% RSLogix 500 project VENTURA PACIFIC 3D_BAK170.RSS, saved by version 11.00.00.00 %
PROJECT "UNTITLED"    % processor: MicroLogix 1400 %

PROGRAM FILES
  LAD 2   213 rungs

DATA FILES
  O0 OUTPUT  7 elements
  I1 INPUT  26 elements
  S2 STATUS  66 elements
  B3 BINARY  10 elements
  T4 TIMER  35 elements  % Moves timing value into Time delay for bin eject %
  C5 COUNTER  9 elements
  R6 CONTROL  1 elements
  N7 INTEGER  33 elements
  F8 FLOAT  3 elements

LADDER 2
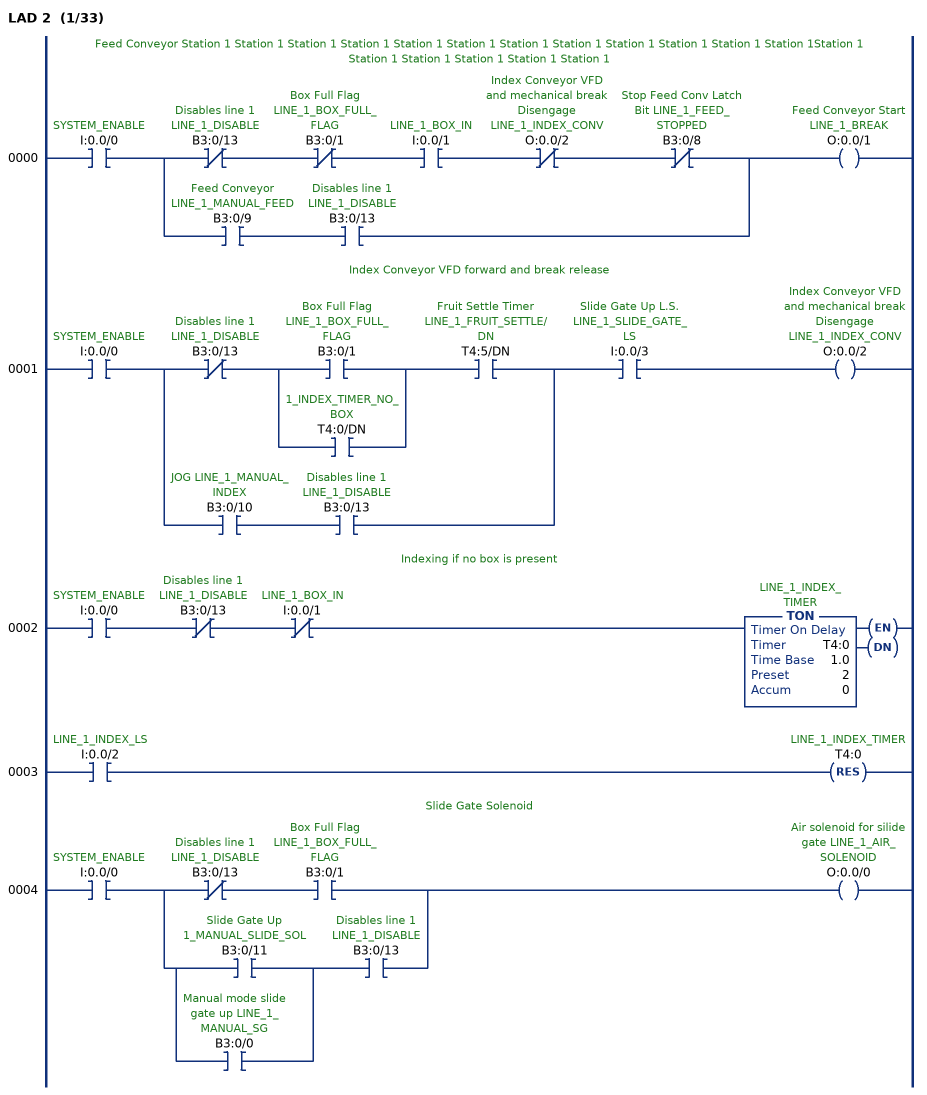
% Rung: 0 %
% Feed Conveyor Station 1 Station 1 Station 1 Station 1 Station 1 Station 1 Station 1 Station 1 Station 1 Station 1 Station 1 Station 1Station 1 Station 1 Station 1 Station 1 Station 1 Station 1 %
SOR XIC I:0.0/0 BST XIO B3:0/13 XIO B3:0/1 XIC I:0.0/1 XIO O:0.0/2 XIO B3:0/8 NXB XIC B3:0/9 XIC B3:0/13 BND OTE O:0.0/1 EOR
%   I:0.0/0  SYSTEM_ENABLE %
%   B3:0/13  LINE_1_DISABLE  "Disables line 1" %
%   B3:0/1  LINE_1_BOX_FULL_FLAG  "Box Full Flag" %
%   I:0.0/1  LINE_1_BOX_IN %
%   O:0.0/2  LINE_1_INDEX_CONV  "Index Conveyor VFD and mechanical break Disengage" %
%   B3:0/8  LINE_1_FEED_STOPPED  "Stop Feed Conv Latch Bit" %
%   B3:0/9  LINE_1_MANUAL_FEED  "Feed Conveyor" %
%   O:0.0/1  LINE_1_BREAK  "Feed Conveyor Start" %
% Rung: 1 %
% Index Conveyor VFD forward and break release %
SOR XIC I:0.0/0 BST XIO B3:0/13 BST XIC B3:0/1 NXB XIC T4:0/DN BND XIC T4:5/DN NXB XIC B3:0/10 XIC B3:0/13 BND XIC I:0.0/3 OTE O:0.0/2 EOR
%   I:0.0/0  SYSTEM_ENABLE %
%   B3:0/13  LINE_1_DISABLE  "Disables line 1" %
%   B3:0/1  LINE_1_BOX_FULL_FLAG  "Box Full Flag" %
%   T4:0/DN  1_INDEX_TIMER_NO_BOX %
%   T4:5  LINE_1_FRUIT_SETTLE  "Fruit Settle Timer" %
%   B3:0/10  LINE_1_MANUAL_INDEX  "JOG" %
%   I:0.0/3  LINE_1_SLIDE_GATE_LS  "Slide Gate Up L.S." %
%   O:0.0/2  LINE_1_INDEX_CONV  "Index Conveyor VFD and mechanical break Disengage" %
% Rung: 2 %
% Indexing if no box is present %
SOR XIC I:0.0/0 XIO B3:0/13 XIO I:0.0/1 TON T4:0 1.0 2 0 EOR
%   I:0.0/0  SYSTEM_ENABLE %
%   B3:0/13  LINE_1_DISABLE  "Disables line 1" %
%   I:0.0/1  LINE_1_BOX_IN %
%   T4:0  LINE_1_INDEX_TIMER %
% Rung: 3 %
SOR XIC I:0.0/2 RES T4:0 EOR
%   I:0.0/2  LINE_1_INDEX_LS %
%   T4:0  LINE_1_INDEX_TIMER %
% Rung: 4 %
% Slide Gate Solenoid %
SOR XIC I:0.0/0 BST XIO B3:0/13 XIC B3:0/1 NXB BST XIC B3:0/11 NXB XIC B3:0/0 BND XIC B3:0/13 BND OTE O:0.0/0 EOR
%   I:0.0/0  SYSTEM_ENABLE %
%   B3:0/13  LINE_1_DISABLE  "Disables line 1" %
%   B3:0/1  LINE_1_BOX_FULL_FLAG  "Box Full Flag" %
%   B3:0/11  1_MANUAL_SLIDE_SOL  "Slide Gate Up" %
%   B3:0/0  LINE_1_MANUAL_SG  "Manual mode slide gate up" %
%   O:0.0/0  LINE_1_AIR_SOLENOID  "Air solenoid for silide gate" %

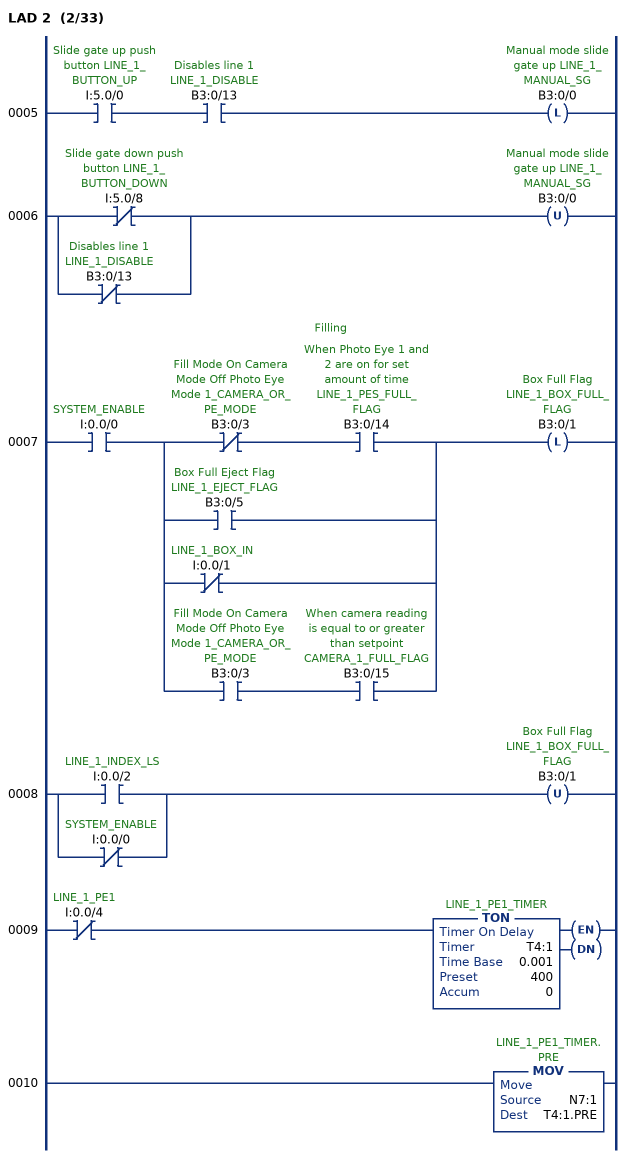
% Rung: 5 %
SOR XIC I:5.0/0 XIC B3:0/13 OTL B3:0/0 EOR
%   I:5.0/0  LINE_1_BUTTON_UP  "Slide gate up push button" %
%   B3:0/13  LINE_1_DISABLE  "Disables line 1" %
%   B3:0/0  LINE_1_MANUAL_SG  "Manual mode slide gate up" %
% Rung: 6 %
SOR BST XIO I:5.0/8 NXB XIO B3:0/13 BND OTU B3:0/0 EOR
%   I:5.0/8  LINE_1_BUTTON_DOWN  "Slide gate down push button" %
%   B3:0/13  LINE_1_DISABLE  "Disables line 1" %
%   B3:0/0  LINE_1_MANUAL_SG  "Manual mode slide gate up" %
% Rung: 7 %
% Filling %
SOR XIC I:0.0/0 BST XIO B3:0/3 XIC B3:0/14 NXB BST XIC B3:0/5 NXB BST XIO I:0.0/1 NXB XIC B3:0/3 XIC B3:0/15 BND BND BND OTL B3:0/1 EOR
%   I:0.0/0  SYSTEM_ENABLE %
%   B3:0/3  1_CAMERA_OR_PE_MODE  "Fill Mode On Camera Mode Off Photo Eye Mode" %
%   B3:0/14  LINE_1_PES_FULL_FLAG  "When Photo Eye 1 and 2 are on for set amount of time" %
%   B3:0/5  LINE_1_EJECT_FLAG  "Box Full Eject Flag" %
%   I:0.0/1  LINE_1_BOX_IN %
%   B3:0/15  CAMERA_1_FULL_FLAG  "When camera reading is equal to or greater than setpoint" %
%   B3:0/1  LINE_1_BOX_FULL_FLAG  "Box Full Flag" %
% Rung: 8 %
SOR BST XIC I:0.0/2 NXB XIO I:0.0/0 BND OTU B3:0/1 EOR
%   I:0.0/2  LINE_1_INDEX_LS %
%   I:0.0/0  SYSTEM_ENABLE %
%   B3:0/1  LINE_1_BOX_FULL_FLAG  "Box Full Flag" %
% Rung: 9 %
SOR XIO I:0.0/4 TON T4:1 0.001 400 0 EOR
%   I:0.0/4  LINE_1_PE1 %
%   T4:1  LINE_1_PE1_TIMER %
% Rung: 10 %
SOR MOV N7:1 T4:1.PRE EOR
%   N7:1  LINE_1_PE1_TIME_MOV %
%   T4:1  LINE_1_PE1_TIMER %

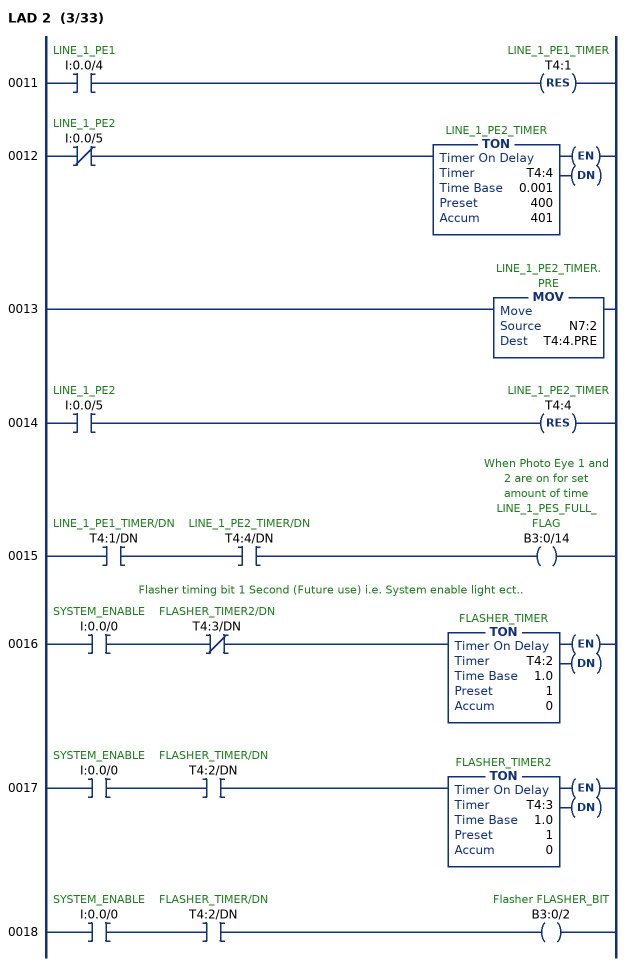
% Rung: 11 %
SOR XIC I:0.0/4 RES T4:1 EOR
%   I:0.0/4  LINE_1_PE1 %
%   T4:1  LINE_1_PE1_TIMER %
% Rung: 12 %
SOR XIO I:0.0/5 TON T4:4 0.001 400 401 EOR
%   I:0.0/5  LINE_1_PE2 %
%   T4:4  LINE_1_PE2_TIMER %
% Rung: 13 %
SOR MOV N7:2 T4:4.PRE EOR
%   N7:2  LINE_1_PE2_TIME_MOV %
%   T4:4  LINE_1_PE2_TIMER %
% Rung: 14 %
SOR XIC I:0.0/5 RES T4:4 EOR
%   I:0.0/5  LINE_1_PE2 %
%   T4:4  LINE_1_PE2_TIMER %
% Rung: 15 %
SOR XIC T4:1/DN XIC T4:4/DN OTE B3:0/14 EOR
%   T4:1  LINE_1_PE1_TIMER %
%   T4:4  LINE_1_PE2_TIMER %
%   B3:0/14  LINE_1_PES_FULL_FLAG  "When Photo Eye 1 and 2 are on for set amount of time" %
% Rung: 16 %
% Flasher timing bit 1 Second (Future use) i.e. System enable light ect.. %
SOR XIC I:0.0/0 XIO T4:3/DN TON T4:2 1.0 1 0 EOR
%   I:0.0/0  SYSTEM_ENABLE %
%   T4:3  FLASHER_TIMER2 %
%   T4:2  FLASHER_TIMER %
% Rung: 17 %
SOR XIC I:0.0/0 XIC T4:2/DN TON T4:3 1.0 1 0 EOR
%   I:0.0/0  SYSTEM_ENABLE %
%   T4:2  FLASHER_TIMER %
%   T4:3  FLASHER_TIMER2 %
% Rung: 18 %
SOR XIC I:0.0/0 XIC T4:2/DN OTE B3:0/2 EOR
%   I:0.0/0  SYSTEM_ENABLE %
%   T4:2  FLASHER_TIMER %
%   B3:0/2  FLASHER_BIT  "Flasher" %

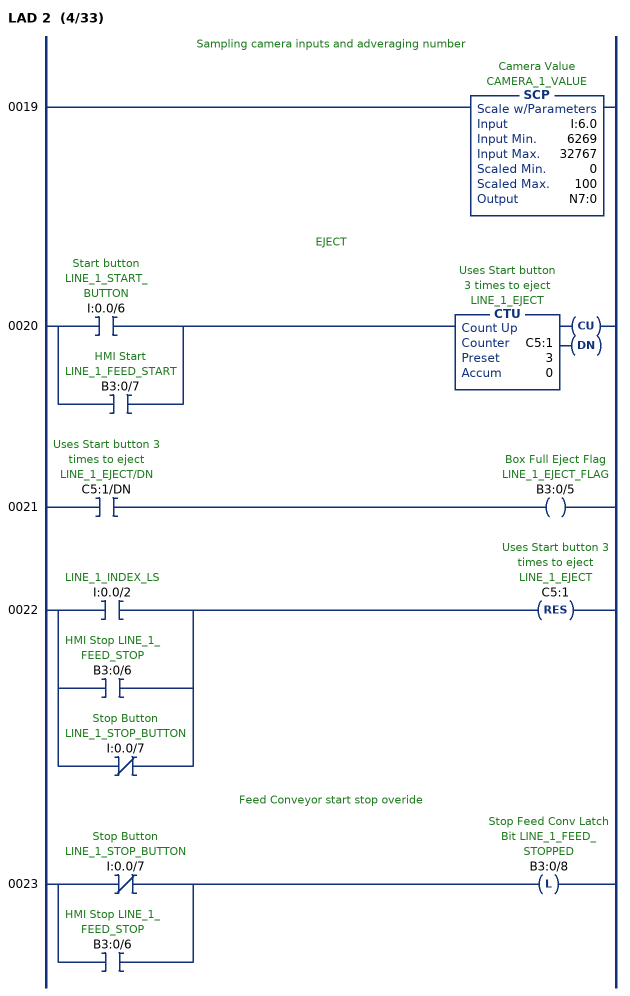
% Rung: 19 %
% Sampling camera inputs and adveraging number %
SOR SCP I:6.0 6269 32767 0 100 N7:0 EOR
%   N7:0  CAMERA_1_VALUE  "Camera Value" %
% Rung: 20 %
% EJECT %
SOR BST XIC I:0.0/6 NXB XIC B3:0/7 BND CTU C5:1 3 0 EOR
%   I:0.0/6  LINE_1_START_BUTTON  "Start button" %
%   B3:0/7  LINE_1_FEED_START  "HMI Start" %
%   C5:1  LINE_1_EJECT  "Uses Start button 3 times to eject" %
% Rung: 21 %
SOR XIC C5:1/DN OTE B3:0/5 EOR
%   C5:1  LINE_1_EJECT  "Uses Start button 3 times to eject" %
%   B3:0/5  LINE_1_EJECT_FLAG  "Box Full Eject Flag" %
% Rung: 22 %
SOR BST XIC I:0.0/2 NXB BST XIC B3:0/6 NXB XIO I:0.0/7 BND BND RES C5:1 EOR
%   I:0.0/2  LINE_1_INDEX_LS %
%   B3:0/6  LINE_1_FEED_STOP  "HMI Stop" %
%   I:0.0/7  LINE_1_STOP_BUTTON  "Stop Button" %
%   C5:1  LINE_1_EJECT  "Uses Start button 3 times to eject" %
% Rung: 23 %
% Feed Conveyor start stop overide %
SOR BST XIO I:0.0/7 NXB XIC B3:0/6 BND OTL B3:0/8 EOR
%   I:0.0/7  LINE_1_STOP_BUTTON  "Stop Button" %
%   B3:0/6  LINE_1_FEED_STOP  "HMI Stop" %
%   B3:0/8  LINE_1_FEED_STOPPED  "Stop Feed Conv Latch Bit" %

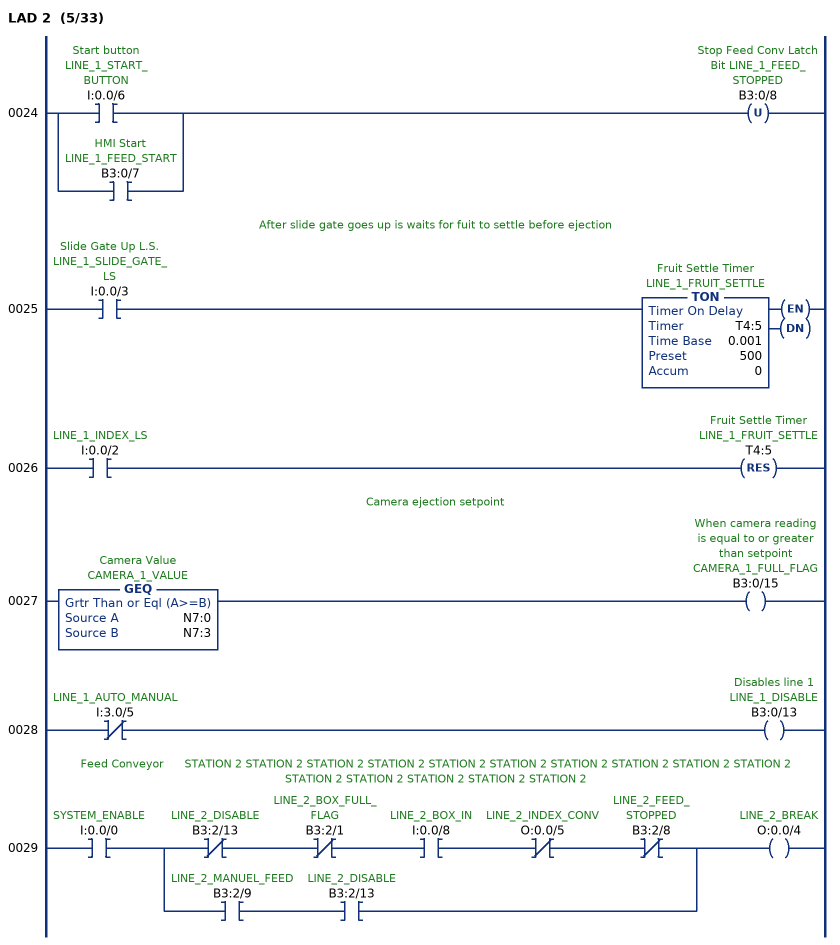
% Rung: 24 %
SOR BST XIC I:0.0/6 NXB XIC B3:0/7 BND OTU B3:0/8 EOR
%   I:0.0/6  LINE_1_START_BUTTON  "Start button" %
%   B3:0/7  LINE_1_FEED_START  "HMI Start" %
%   B3:0/8  LINE_1_FEED_STOPPED  "Stop Feed Conv Latch Bit" %
% Rung: 25 %
% After slide gate goes up is waits for fuit to settle before ejection %
SOR XIC I:0.0/3 TON T4:5 0.001 500 0 EOR
%   I:0.0/3  LINE_1_SLIDE_GATE_LS  "Slide Gate Up L.S." %
%   T4:5  LINE_1_FRUIT_SETTLE  "Fruit Settle Timer" %
% Rung: 26 %
SOR XIC I:0.0/2 RES T4:5 EOR
%   I:0.0/2  LINE_1_INDEX_LS %
%   T4:5  LINE_1_FRUIT_SETTLE  "Fruit Settle Timer" %
% Rung: 27 %
% Camera ejection setpoint %
SOR GEQ N7:0 N7:3 OTE B3:0/15 EOR
%   N7:0  CAMERA_1_VALUE  "Camera Value" %
%   N7:3  LINE_1_CAMERA_EJECT %
%   B3:0/15  CAMERA_1_FULL_FLAG  "When camera reading is equal to or greater than setpoint" %
% Rung: 28 %
SOR XIO I:3.0/5 OTE B3:0/13 EOR
%   I:3.0/5  LINE_1_AUTO_MANUAL %
%   B3:0/13  LINE_1_DISABLE  "Disables line 1" %
% Rung: 29 %
% Feed Conveyor      STATION 2 STATION 2 STATION 2 STATION 2 STATION 2 STATION 2 STATION 2 STATION 2 STATION 2 STATION 2 STATION 2 STATION 2 STATION 2 STATION 2 STATION 2 %
SOR XIC I:0.0/0 BST XIO B3:2/13 XIO B3:2/1 XIC I:0.0/8 XIO O:0.0/5 XIO B3:2/8 NXB XIC B3:2/9 XIC B3:2/13 BND OTE O:0.0/4 EOR
%   I:0.0/0  SYSTEM_ENABLE %
%   B3:2/13  LINE_2_DISABLE %
%   B3:2/1  LINE_2_BOX_FULL_FLAG %
%   I:0.0/8  LINE_2_BOX_IN %
%   O:0.0/5  LINE_2_INDEX_CONV %
%   B3:2/8  LINE_2_FEED_STOPPED %
%   B3:2/9  LINE_2_MANUEL_FEED %
%   O:0.0/4  LINE_2_BREAK %

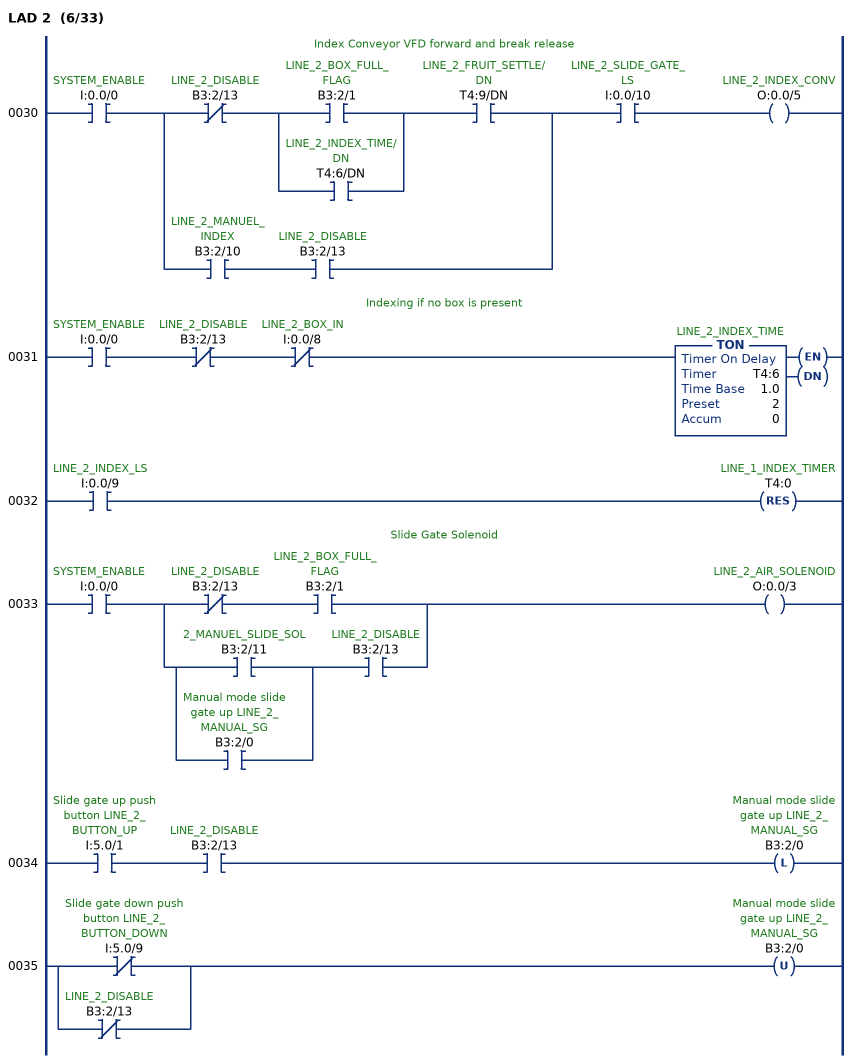
% Rung: 30 %
% Index Conveyor VFD forward and break release %
SOR XIC I:0.0/0 BST XIO B3:2/13 BST XIC B3:2/1 NXB XIC T4:6/DN BND XIC T4:9/DN NXB XIC B3:2/10 XIC B3:2/13 BND XIC I:0.0/10 OTE O:0.0/5 EOR
%   I:0.0/0  SYSTEM_ENABLE %
%   B3:2/13  LINE_2_DISABLE %
%   B3:2/1  LINE_2_BOX_FULL_FLAG %
%   T4:6  LINE_2_INDEX_TIME %
%   T4:9  LINE_2_FRUIT_SETTLE %
%   B3:2/10  LINE_2_MANUEL_INDEX %
%   I:0.0/10  LINE_2_SLIDE_GATE_LS %
%   O:0.0/5  LINE_2_INDEX_CONV %
% Rung: 31 %
% Indexing if no box is present %
SOR XIC I:0.0/0 XIO B3:2/13 XIO I:0.0/8 TON T4:6 1.0 2 0 EOR
%   I:0.0/0  SYSTEM_ENABLE %
%   B3:2/13  LINE_2_DISABLE %
%   I:0.0/8  LINE_2_BOX_IN %
%   T4:6  LINE_2_INDEX_TIME %
% Rung: 32 %
SOR XIC I:0.0/9 RES T4:0 EOR
%   I:0.0/9  LINE_2_INDEX_LS %
%   T4:0  LINE_1_INDEX_TIMER %
% Rung: 33 %
% Slide Gate Solenoid %
SOR XIC I:0.0/0 BST XIO B3:2/13 XIC B3:2/1 NXB BST XIC B3:2/11 NXB XIC B3:2/0 BND XIC B3:2/13 BND OTE O:0.0/3 EOR
%   I:0.0/0  SYSTEM_ENABLE %
%   B3:2/13  LINE_2_DISABLE %
%   B3:2/1  LINE_2_BOX_FULL_FLAG %
%   B3:2/11  2_MANUEL_SLIDE_SOL %
%   B3:2/0  LINE_2_MANUAL_SG  "Manual mode slide gate up" %
%   O:0.0/3  LINE_2_AIR_SOLENOID %
% Rung: 34 %
SOR XIC I:5.0/1 XIC B3:2/13 OTL B3:2/0 EOR
%   I:5.0/1  LINE_2_BUTTON_UP  "Slide gate up push button" %
%   B3:2/13  LINE_2_DISABLE %
%   B3:2/0  LINE_2_MANUAL_SG  "Manual mode slide gate up" %
% Rung: 35 %
SOR BST XIO I:5.0/9 NXB XIO B3:2/13 BND OTU B3:2/0 EOR
%   I:5.0/9  LINE_2_BUTTON_DOWN  "Slide gate down push button" %
%   B3:2/13  LINE_2_DISABLE %
%   B3:2/0  LINE_2_MANUAL_SG  "Manual mode slide gate up" %

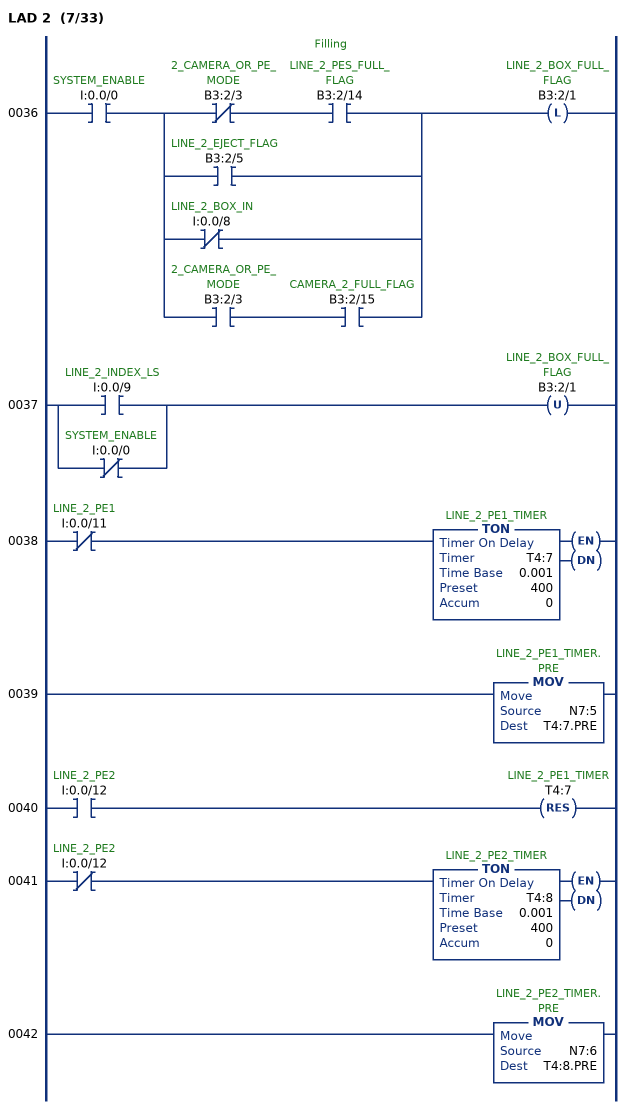
% Rung: 36 %
% Filling %
SOR XIC I:0.0/0 BST XIO B3:2/3 XIC B3:2/14 NXB BST XIC B3:2/5 NXB BST XIO I:0.0/8 NXB XIC B3:2/3 XIC B3:2/15 BND BND BND OTL B3:2/1 EOR
%   I:0.0/0  SYSTEM_ENABLE %
%   B3:2/3  2_CAMERA_OR_PE_MODE %
%   B3:2/14  LINE_2_PES_FULL_FLAG %
%   B3:2/5  LINE_2_EJECT_FLAG %
%   I:0.0/8  LINE_2_BOX_IN %
%   B3:2/15  CAMERA_2_FULL_FLAG %
%   B3:2/1  LINE_2_BOX_FULL_FLAG %
% Rung: 37 %
SOR BST XIC I:0.0/9 NXB XIO I:0.0/0 BND OTU B3:2/1 EOR
%   I:0.0/9  LINE_2_INDEX_LS %
%   I:0.0/0  SYSTEM_ENABLE %
%   B3:2/1  LINE_2_BOX_FULL_FLAG %
% Rung: 38 %
SOR XIO I:0.0/11 TON T4:7 0.001 400 0 EOR
%   I:0.0/11  LINE_2_PE1 %
%   T4:7  LINE_2_PE1_TIMER %
% Rung: 39 %
SOR MOV N7:5 T4:7.PRE EOR
%   N7:5  LINE_2_PE1_TIME_MOV %
%   T4:7  LINE_2_PE1_TIMER %
% Rung: 40 %
SOR XIC I:0.0/12 RES T4:7 EOR
%   I:0.0/12  LINE_2_PE2 %
%   T4:7  LINE_2_PE1_TIMER %
% Rung: 41 %
SOR XIO I:0.0/12 TON T4:8 0.001 400 0 EOR
%   I:0.0/12  LINE_2_PE2 %
%   T4:8  LINE_2_PE2_TIMER %
% Rung: 42 %
SOR MOV N7:6 T4:8.PRE EOR
%   N7:6  LINE_2_PE2_TIME_MOV %
%   T4:8  LINE_2_PE2_TIMER %

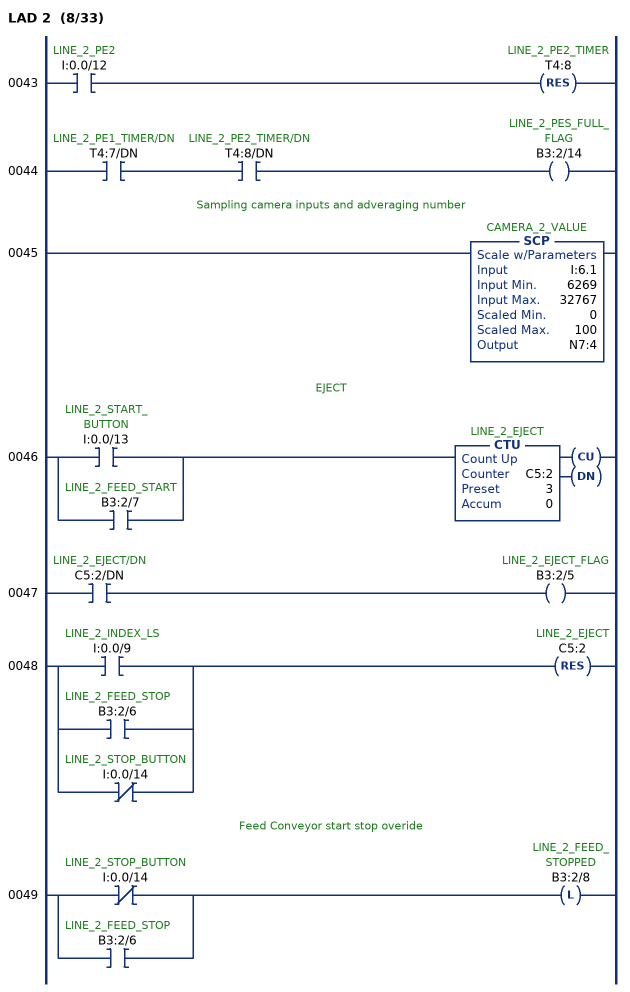
% Rung: 43 %
SOR XIC I:0.0/12 RES T4:8 EOR
%   I:0.0/12  LINE_2_PE2 %
%   T4:8  LINE_2_PE2_TIMER %
% Rung: 44 %
SOR XIC T4:7/DN XIC T4:8/DN OTE B3:2/14 EOR
%   T4:7  LINE_2_PE1_TIMER %
%   T4:8  LINE_2_PE2_TIMER %
%   B3:2/14  LINE_2_PES_FULL_FLAG %
% Rung: 45 %
% Sampling camera inputs and adveraging number %
SOR SCP I:6.1 6269 32767 0 100 N7:4 EOR
%   N7:4  CAMERA_2_VALUE %
% Rung: 46 %
% EJECT %
SOR BST XIC I:0.0/13 NXB XIC B3:2/7 BND CTU C5:2 3 0 EOR
%   I:0.0/13  LINE_2_START_BUTTON %
%   B3:2/7  LINE_2_FEED_START %
%   C5:2  LINE_2_EJECT %
% Rung: 47 %
SOR XIC C5:2/DN OTE B3:2/5 EOR
%   C5:2  LINE_2_EJECT %
%   B3:2/5  LINE_2_EJECT_FLAG %
% Rung: 48 %
SOR BST XIC I:0.0/9 NXB BST XIC B3:2/6 NXB XIO I:0.0/14 BND BND RES C5:2 EOR
%   I:0.0/9  LINE_2_INDEX_LS %
%   B3:2/6  LINE_2_FEED_STOP %
%   I:0.0/14  LINE_2_STOP_BUTTON %
%   C5:2  LINE_2_EJECT %
% Rung: 49 %
% Feed Conveyor start stop overide %
SOR BST XIO I:0.0/14 NXB XIC B3:2/6 BND OTL B3:2/8 EOR
%   I:0.0/14  LINE_2_STOP_BUTTON %
%   B3:2/6  LINE_2_FEED_STOP %
%   B3:2/8  LINE_2_FEED_STOPPED %

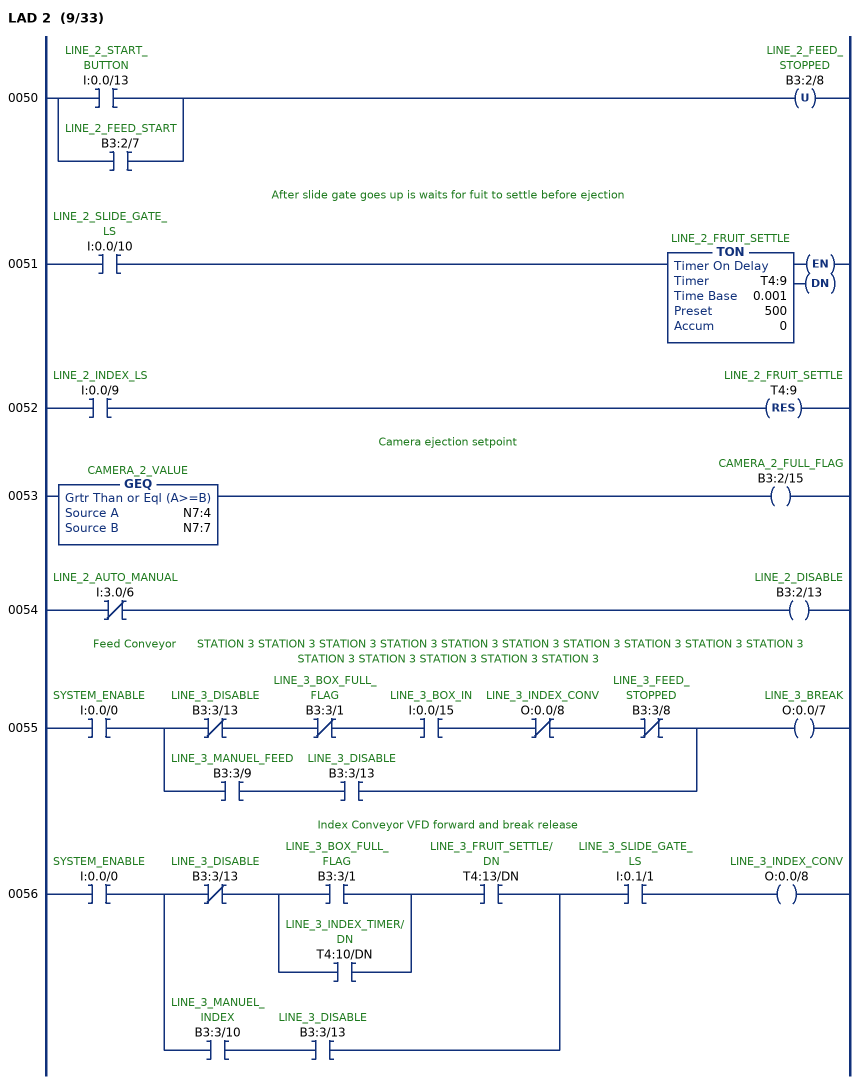
% Rung: 50 %
SOR BST XIC I:0.0/13 NXB XIC B3:2/7 BND OTU B3:2/8 EOR
%   I:0.0/13  LINE_2_START_BUTTON %
%   B3:2/7  LINE_2_FEED_START %
%   B3:2/8  LINE_2_FEED_STOPPED %
% Rung: 51 %
% After slide gate goes up is waits for fuit to settle before ejection %
SOR XIC I:0.0/10 TON T4:9 0.001 500 0 EOR
%   I:0.0/10  LINE_2_SLIDE_GATE_LS %
%   T4:9  LINE_2_FRUIT_SETTLE %
% Rung: 52 %
SOR XIC I:0.0/9 RES T4:9 EOR
%   I:0.0/9  LINE_2_INDEX_LS %
%   T4:9  LINE_2_FRUIT_SETTLE %
% Rung: 53 %
% Camera ejection setpoint %
SOR GEQ N7:4 N7:7 OTE B3:2/15 EOR
%   N7:4  CAMERA_2_VALUE %
%   N7:7  LINE_2_CAMERA_EJECT %
%   B3:2/15  CAMERA_2_FULL_FLAG %
% Rung: 54 %
SOR XIO I:3.0/6 OTE B3:2/13 EOR
%   I:3.0/6  LINE_2_AUTO_MANUAL %
%   B3:2/13  LINE_2_DISABLE %
% Rung: 55 %
% Feed Conveyor      STATION 3 STATION 3 STATION 3 STATION 3 STATION 3 STATION 3 STATION 3 STATION 3 STATION 3 STATION 3 STATION 3 STATION 3 STATION 3 STATION 3 STATION 3 %
SOR XIC I:0.0/0 BST XIO B3:3/13 XIO B3:3/1 XIC I:0.0/15 XIO O:0.0/8 XIO B3:3/8 NXB XIC B3:3/9 XIC B3:3/13 BND OTE O:0.0/7 EOR
%   I:0.0/0  SYSTEM_ENABLE %
%   B3:3/13  LINE_3_DISABLE %
%   B3:3/1  LINE_3_BOX_FULL_FLAG %
%   I:0.0/15  LINE_3_BOX_IN %
%   O:0.0/8  LINE_3_INDEX_CONV %
%   B3:3/8  LINE_3_FEED_STOPPED %
%   B3:3/9  LINE_3_MANUEL_FEED %
%   O:0.0/7  LINE_3_BREAK %
% Rung: 56 %
% Index Conveyor VFD forward and break release %
SOR XIC I:0.0/0 BST XIO B3:3/13 BST XIC B3:3/1 NXB XIC T4:10/DN BND XIC T4:13/DN NXB XIC B3:3/10 XIC B3:3/13 BND XIC I:0.1/1 OTE O:0.0/8 EOR
%   I:0.0/0  SYSTEM_ENABLE %
%   B3:3/13  LINE_3_DISABLE %
%   B3:3/1  LINE_3_BOX_FULL_FLAG %
%   T4:10  LINE_3_INDEX_TIMER %
%   T4:13  LINE_3_FRUIT_SETTLE %
%   B3:3/10  LINE_3_MANUEL_INDEX %
%   I:0.1/1  LINE_3_SLIDE_GATE_LS %
%   O:0.0/8  LINE_3_INDEX_CONV %

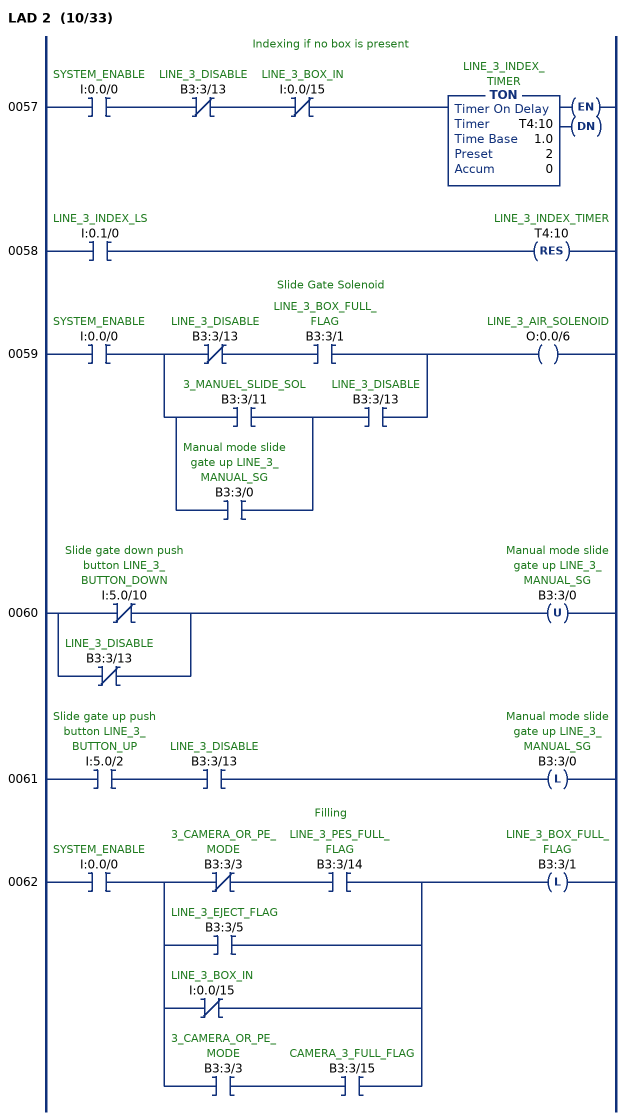
% Rung: 57 %
% Indexing if no box is present %
SOR XIC I:0.0/0 XIO B3:3/13 XIO I:0.0/15 TON T4:10 1.0 2 0 EOR
%   I:0.0/0  SYSTEM_ENABLE %
%   B3:3/13  LINE_3_DISABLE %
%   I:0.0/15  LINE_3_BOX_IN %
%   T4:10  LINE_3_INDEX_TIMER %
% Rung: 58 %
SOR XIC I:0.1/0 RES T4:10 EOR
%   I:0.1/0  LINE_3_INDEX_LS %
%   T4:10  LINE_3_INDEX_TIMER %
% Rung: 59 %
% Slide Gate Solenoid %
SOR XIC I:0.0/0 BST XIO B3:3/13 XIC B3:3/1 NXB BST XIC B3:3/11 NXB XIC B3:3/0 BND XIC B3:3/13 BND OTE O:0.0/6 EOR
%   I:0.0/0  SYSTEM_ENABLE %
%   B3:3/13  LINE_3_DISABLE %
%   B3:3/1  LINE_3_BOX_FULL_FLAG %
%   B3:3/11  3_MANUEL_SLIDE_SOL %
%   B3:3/0  LINE_3_MANUAL_SG  "Manual mode slide gate up" %
%   O:0.0/6  LINE_3_AIR_SOLENOID %
% Rung: 60 %
SOR BST XIO I:5.0/10 NXB XIO B3:3/13 BND OTU B3:3/0 EOR
%   I:5.0/10  LINE_3_BUTTON_DOWN  "Slide gate down push button" %
%   B3:3/13  LINE_3_DISABLE %
%   B3:3/0  LINE_3_MANUAL_SG  "Manual mode slide gate up" %
% Rung: 61 %
SOR XIC I:5.0/2 XIC B3:3/13 OTL B3:3/0 EOR
%   I:5.0/2  LINE_3_BUTTON_UP  "Slide gate up push button" %
%   B3:3/13  LINE_3_DISABLE %
%   B3:3/0  LINE_3_MANUAL_SG  "Manual mode slide gate up" %
% Rung: 62 %
% Filling %
SOR XIC I:0.0/0 BST XIO B3:3/3 XIC B3:3/14 NXB BST XIC B3:3/5 NXB BST XIO I:0.0/15 NXB XIC B3:3/3 XIC B3:3/15 BND BND BND OTL B3:3/1 EOR
%   I:0.0/0  SYSTEM_ENABLE %
%   B3:3/3  3_CAMERA_OR_PE_MODE %
%   B3:3/14  LINE_3_PES_FULL_FLAG %
%   B3:3/5  LINE_3_EJECT_FLAG %
%   I:0.0/15  LINE_3_BOX_IN %
%   B3:3/15  CAMERA_3_FULL_FLAG %
%   B3:3/1  LINE_3_BOX_FULL_FLAG %

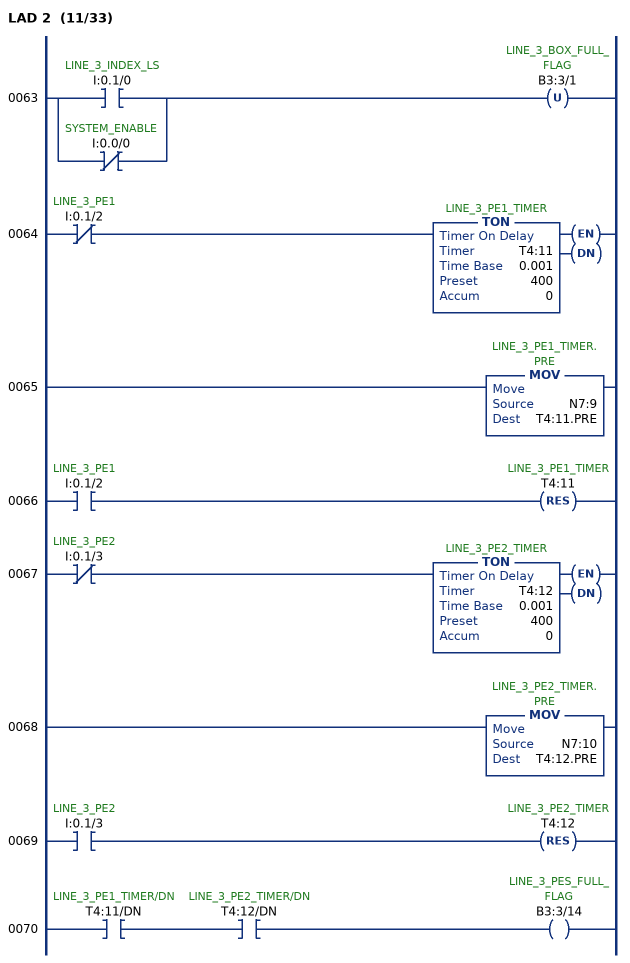
% Rung: 63 %
SOR BST XIC I:0.1/0 NXB XIO I:0.0/0 BND OTU B3:3/1 EOR
%   I:0.1/0  LINE_3_INDEX_LS %
%   I:0.0/0  SYSTEM_ENABLE %
%   B3:3/1  LINE_3_BOX_FULL_FLAG %
% Rung: 64 %
SOR XIO I:0.1/2 TON T4:11 0.001 400 0 EOR
%   I:0.1/2  LINE_3_PE1 %
%   T4:11  LINE_3_PE1_TIMER %
% Rung: 65 %
SOR MOV N7:9 T4:11.PRE EOR
%   N7:9  LINE_3_PE1_TIME_MOV %
%   T4:11  LINE_3_PE1_TIMER %
% Rung: 66 %
SOR XIC I:0.1/2 RES T4:11 EOR
%   I:0.1/2  LINE_3_PE1 %
%   T4:11  LINE_3_PE1_TIMER %
% Rung: 67 %
SOR XIO I:0.1/3 TON T4:12 0.001 400 0 EOR
%   I:0.1/3  LINE_3_PE2 %
%   T4:12  LINE_3_PE2_TIMER %
% Rung: 68 %
SOR MOV N7:10 T4:12.PRE EOR
%   N7:10  LINE_3_PE2_TIME_MOV %
%   T4:12  LINE_3_PE2_TIMER %
% Rung: 69 %
SOR XIC I:0.1/3 RES T4:12 EOR
%   I:0.1/3  LINE_3_PE2 %
%   T4:12  LINE_3_PE2_TIMER %
% Rung: 70 %
SOR XIC T4:11/DN XIC T4:12/DN OTE B3:3/14 EOR
%   T4:11  LINE_3_PE1_TIMER %
%   T4:12  LINE_3_PE2_TIMER %
%   B3:3/14  LINE_3_PES_FULL_FLAG %

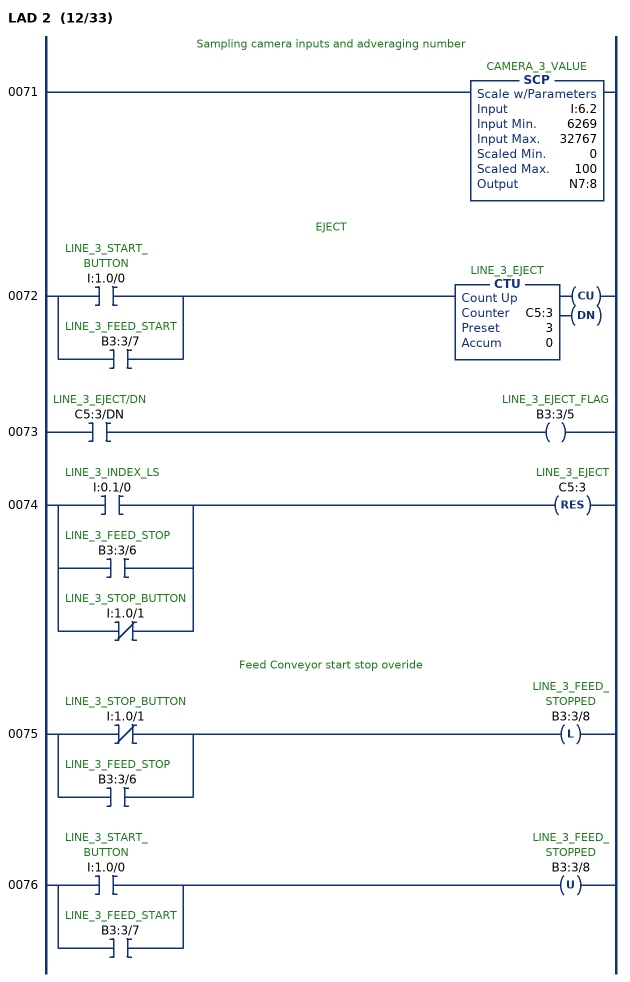
% Rung: 71 %
% Sampling camera inputs and adveraging number %
SOR SCP I:6.2 6269 32767 0 100 N7:8 EOR
%   N7:8  CAMERA_3_VALUE %
% Rung: 72 %
% EJECT %
SOR BST XIC I:1.0/0 NXB XIC B3:3/7 BND CTU C5:3 3 0 EOR
%   I:1.0/0  LINE_3_START_BUTTON %
%   B3:3/7  LINE_3_FEED_START %
%   C5:3  LINE_3_EJECT %
% Rung: 73 %
SOR XIC C5:3/DN OTE B3:3/5 EOR
%   C5:3  LINE_3_EJECT %
%   B3:3/5  LINE_3_EJECT_FLAG %
% Rung: 74 %
SOR BST XIC I:0.1/0 NXB BST XIC B3:3/6 NXB XIO I:1.0/1 BND BND RES C5:3 EOR
%   I:0.1/0  LINE_3_INDEX_LS %
%   B3:3/6  LINE_3_FEED_STOP %
%   I:1.0/1  LINE_3_STOP_BUTTON %
%   C5:3  LINE_3_EJECT %
% Rung: 75 %
% Feed Conveyor start stop overide %
SOR BST XIO I:1.0/1 NXB XIC B3:3/6 BND OTL B3:3/8 EOR
%   I:1.0/1  LINE_3_STOP_BUTTON %
%   B3:3/6  LINE_3_FEED_STOP %
%   B3:3/8  LINE_3_FEED_STOPPED %
% Rung: 76 %
SOR BST XIC I:1.0/0 NXB XIC B3:3/7 BND OTU B3:3/8 EOR
%   I:1.0/0  LINE_3_START_BUTTON %
%   B3:3/7  LINE_3_FEED_START %
%   B3:3/8  LINE_3_FEED_STOPPED %

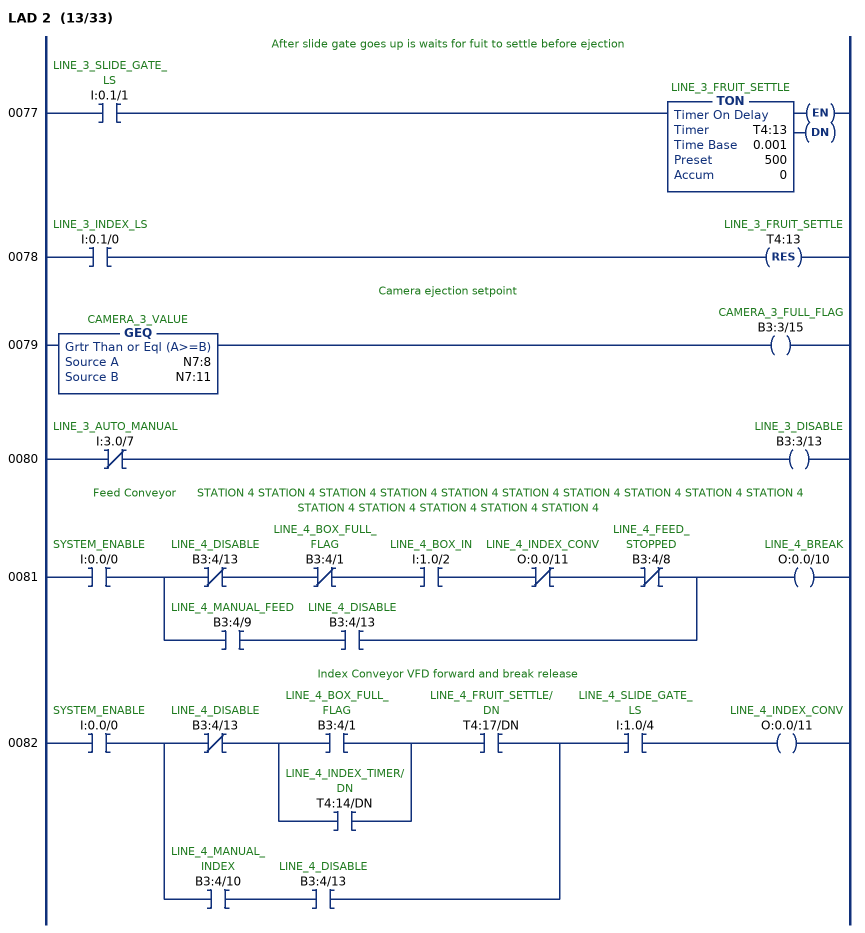
% Rung: 77 %
% After slide gate goes up is waits for fuit to settle before ejection %
SOR XIC I:0.1/1 TON T4:13 0.001 500 0 EOR
%   I:0.1/1  LINE_3_SLIDE_GATE_LS %
%   T4:13  LINE_3_FRUIT_SETTLE %
% Rung: 78 %
SOR XIC I:0.1/0 RES T4:13 EOR
%   I:0.1/0  LINE_3_INDEX_LS %
%   T4:13  LINE_3_FRUIT_SETTLE %
% Rung: 79 %
% Camera ejection setpoint %
SOR GEQ N7:8 N7:11 OTE B3:3/15 EOR
%   N7:8  CAMERA_3_VALUE %
%   N7:11  LINE_3_CAMERA_EJECT %
%   B3:3/15  CAMERA_3_FULL_FLAG %
% Rung: 80 %
SOR XIO I:3.0/7 OTE B3:3/13 EOR
%   I:3.0/7  LINE_3_AUTO_MANUAL %
%   B3:3/13  LINE_3_DISABLE %
% Rung: 81 %
% Feed Conveyor      STATION 4 STATION 4 STATION 4 STATION 4 STATION 4 STATION 4 STATION 4 STATION 4 STATION 4 STATION 4 STATION 4 STATION 4 STATION 4 STATION 4 STATION 4 %
SOR XIC I:0.0/0 BST XIO B3:4/13 XIO B3:4/1 XIC I:1.0/2 XIO O:0.0/11 XIO B3:4/8 NXB XIC B3:4/9 XIC B3:4/13 BND OTE O:0.0/10 EOR
%   I:0.0/0  SYSTEM_ENABLE %
%   B3:4/13  LINE_4_DISABLE %
%   B3:4/1  LINE_4_BOX_FULL_FLAG %
%   I:1.0/2  LINE_4_BOX_IN %
%   O:0.0/11  LINE_4_INDEX_CONV %
%   B3:4/8  LINE_4_FEED_STOPPED %
%   B3:4/9  LINE_4_MANUAL_FEED %
%   O:0.0/10  LINE_4_BREAK %
% Rung: 82 %
% Index Conveyor VFD forward and break release %
SOR XIC I:0.0/0 BST XIO B3:4/13 BST XIC B3:4/1 NXB XIC T4:14/DN BND XIC T4:17/DN NXB XIC B3:4/10 XIC B3:4/13 BND XIC I:1.0/4 OTE O:0.0/11 EOR
%   I:0.0/0  SYSTEM_ENABLE %
%   B3:4/13  LINE_4_DISABLE %
%   B3:4/1  LINE_4_BOX_FULL_FLAG %
%   T4:14  LINE_4_INDEX_TIMER %
%   T4:17  LINE_4_FRUIT_SETTLE %
%   B3:4/10  LINE_4_MANUAL_INDEX %
%   I:1.0/4  LINE_4_SLIDE_GATE_LS %
%   O:0.0/11  LINE_4_INDEX_CONV %

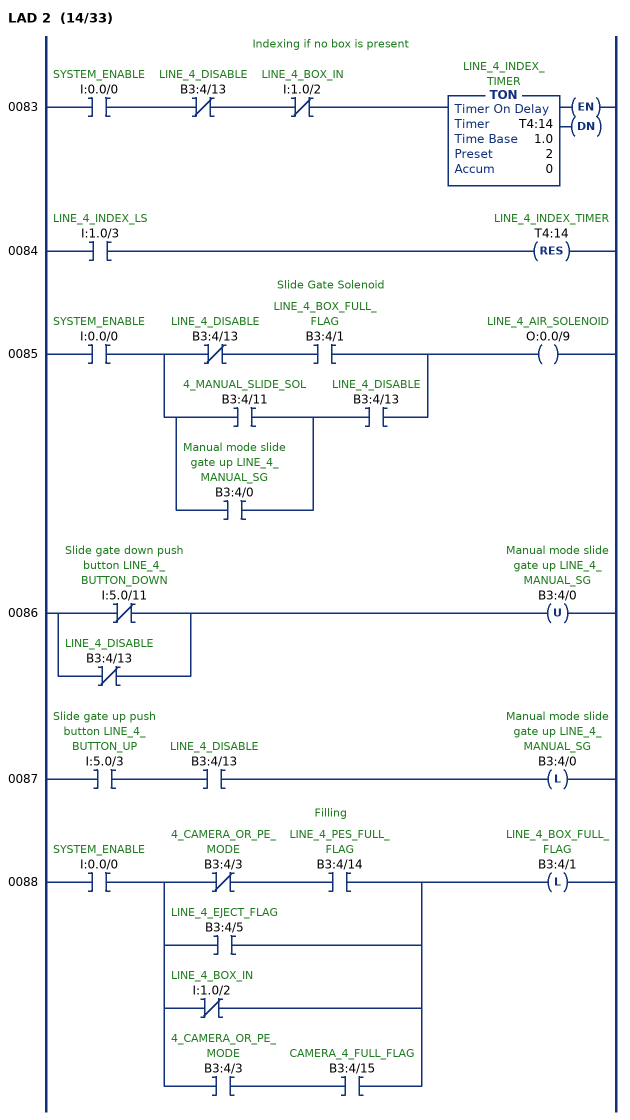
% Rung: 83 %
% Indexing if no box is present %
SOR XIC I:0.0/0 XIO B3:4/13 XIO I:1.0/2 TON T4:14 1.0 2 0 EOR
%   I:0.0/0  SYSTEM_ENABLE %
%   B3:4/13  LINE_4_DISABLE %
%   I:1.0/2  LINE_4_BOX_IN %
%   T4:14  LINE_4_INDEX_TIMER %
% Rung: 84 %
SOR XIC I:1.0/3 RES T4:14 EOR
%   I:1.0/3  LINE_4_INDEX_LS %
%   T4:14  LINE_4_INDEX_TIMER %
% Rung: 85 %
% Slide Gate Solenoid %
SOR XIC I:0.0/0 BST XIO B3:4/13 XIC B3:4/1 NXB BST XIC B3:4/11 NXB XIC B3:4/0 BND XIC B3:4/13 BND OTE O:0.0/9 EOR
%   I:0.0/0  SYSTEM_ENABLE %
%   B3:4/13  LINE_4_DISABLE %
%   B3:4/1  LINE_4_BOX_FULL_FLAG %
%   B3:4/11  4_MANUAL_SLIDE_SOL %
%   B3:4/0  LINE_4_MANUAL_SG  "Manual mode slide gate up" %
%   O:0.0/9  LINE_4_AIR_SOLENOID %
% Rung: 86 %
SOR BST XIO I:5.0/11 NXB XIO B3:4/13 BND OTU B3:4/0 EOR
%   I:5.0/11  LINE_4_BUTTON_DOWN  "Slide gate down push button" %
%   B3:4/13  LINE_4_DISABLE %
%   B3:4/0  LINE_4_MANUAL_SG  "Manual mode slide gate up" %
% Rung: 87 %
SOR XIC I:5.0/3 XIC B3:4/13 OTL B3:4/0 EOR
%   I:5.0/3  LINE_4_BUTTON_UP  "Slide gate up push button" %
%   B3:4/13  LINE_4_DISABLE %
%   B3:4/0  LINE_4_MANUAL_SG  "Manual mode slide gate up" %
% Rung: 88 %
% Filling %
SOR XIC I:0.0/0 BST XIO B3:4/3 XIC B3:4/14 NXB BST XIC B3:4/5 NXB BST XIO I:1.0/2 NXB XIC B3:4/3 XIC B3:4/15 BND BND BND OTL B3:4/1 EOR
%   I:0.0/0  SYSTEM_ENABLE %
%   B3:4/3  4_CAMERA_OR_PE_MODE %
%   B3:4/14  LINE_4_PES_FULL_FLAG %
%   B3:4/5  LINE_4_EJECT_FLAG %
%   I:1.0/2  LINE_4_BOX_IN %
%   B3:4/15  CAMERA_4_FULL_FLAG %
%   B3:4/1  LINE_4_BOX_FULL_FLAG %

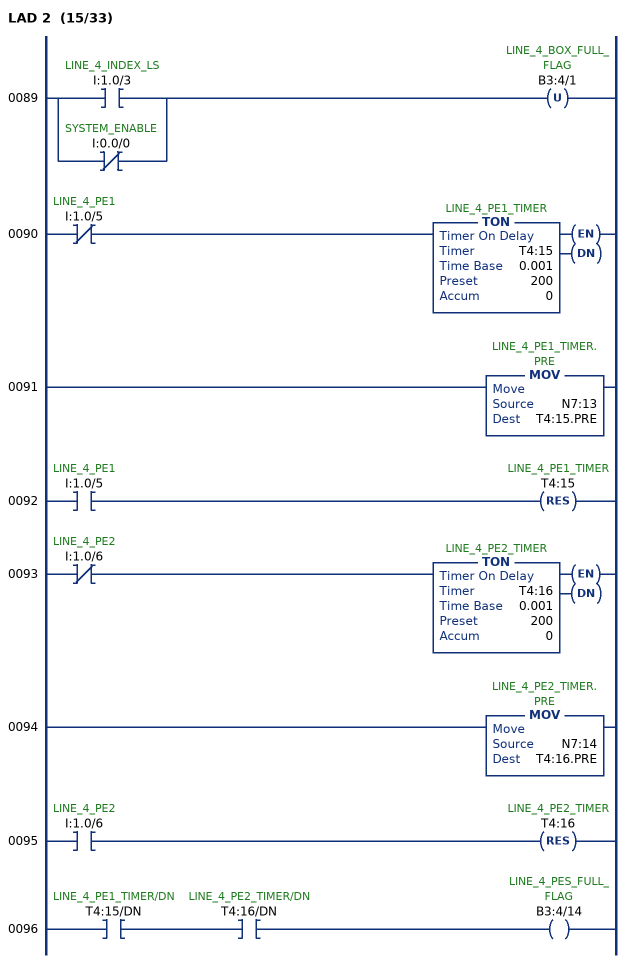
% Rung: 89 %
SOR BST XIC I:1.0/3 NXB XIO I:0.0/0 BND OTU B3:4/1 EOR
%   I:1.0/3  LINE_4_INDEX_LS %
%   I:0.0/0  SYSTEM_ENABLE %
%   B3:4/1  LINE_4_BOX_FULL_FLAG %
% Rung: 90 %
SOR XIO I:1.0/5 TON T4:15 0.001 200 0 EOR
%   I:1.0/5  LINE_4_PE1 %
%   T4:15  LINE_4_PE1_TIMER %
% Rung: 91 %
SOR MOV N7:13 T4:15.PRE EOR
%   N7:13  LINE_4_PE1_TIME_MOV %
%   T4:15  LINE_4_PE1_TIMER %
% Rung: 92 %
SOR XIC I:1.0/5 RES T4:15 EOR
%   I:1.0/5  LINE_4_PE1 %
%   T4:15  LINE_4_PE1_TIMER %
% Rung: 93 %
SOR XIO I:1.0/6 TON T4:16 0.001 200 0 EOR
%   I:1.0/6  LINE_4_PE2 %
%   T4:16  LINE_4_PE2_TIMER %
% Rung: 94 %
SOR MOV N7:14 T4:16.PRE EOR
%   N7:14  LINE_4_PE2_TIME_MOV %
%   T4:16  LINE_4_PE2_TIMER %
% Rung: 95 %
SOR XIC I:1.0/6 RES T4:16 EOR
%   I:1.0/6  LINE_4_PE2 %
%   T4:16  LINE_4_PE2_TIMER %
% Rung: 96 %
SOR XIC T4:15/DN XIC T4:16/DN OTE B3:4/14 EOR
%   T4:15  LINE_4_PE1_TIMER %
%   T4:16  LINE_4_PE2_TIMER %
%   B3:4/14  LINE_4_PES_FULL_FLAG %

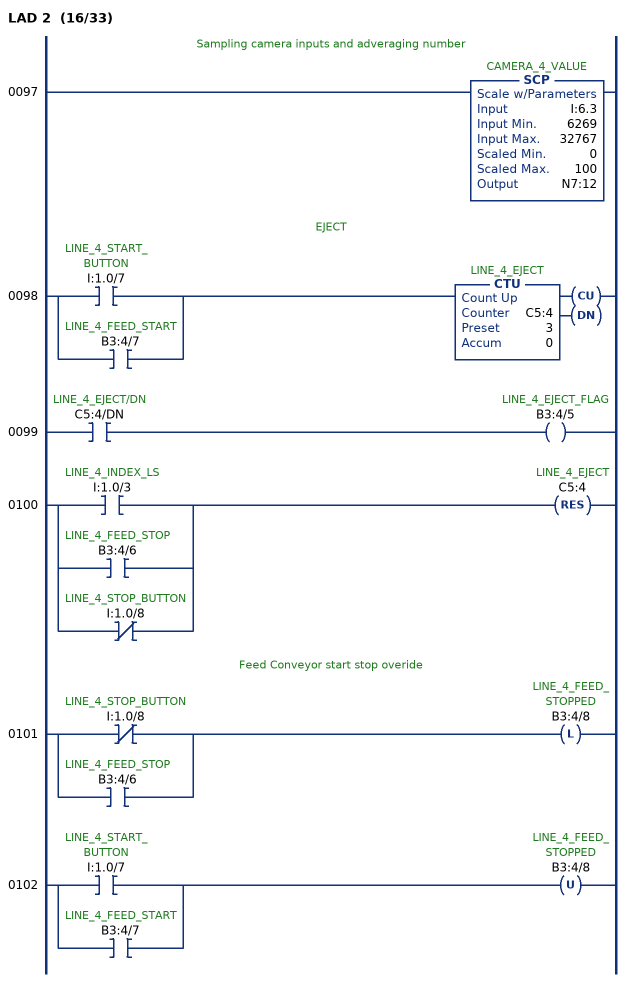
% Rung: 97 %
% Sampling camera inputs and adveraging number %
SOR SCP I:6.3 6269 32767 0 100 N7:12 EOR
%   N7:12  CAMERA_4_VALUE %
% Rung: 98 %
% EJECT %
SOR BST XIC I:1.0/7 NXB XIC B3:4/7 BND CTU C5:4 3 0 EOR
%   I:1.0/7  LINE_4_START_BUTTON %
%   B3:4/7  LINE_4_FEED_START %
%   C5:4  LINE_4_EJECT %
% Rung: 99 %
SOR XIC C5:4/DN OTE B3:4/5 EOR
%   C5:4  LINE_4_EJECT %
%   B3:4/5  LINE_4_EJECT_FLAG %
% Rung: 100 %
SOR BST XIC I:1.0/3 NXB BST XIC B3:4/6 NXB XIO I:1.0/8 BND BND RES C5:4 EOR
%   I:1.0/3  LINE_4_INDEX_LS %
%   B3:4/6  LINE_4_FEED_STOP %
%   I:1.0/8  LINE_4_STOP_BUTTON %
%   C5:4  LINE_4_EJECT %
% Rung: 101 %
% Feed Conveyor start stop overide %
SOR BST XIO I:1.0/8 NXB XIC B3:4/6 BND OTL B3:4/8 EOR
%   I:1.0/8  LINE_4_STOP_BUTTON %
%   B3:4/6  LINE_4_FEED_STOP %
%   B3:4/8  LINE_4_FEED_STOPPED %
% Rung: 102 %
SOR BST XIC I:1.0/7 NXB XIC B3:4/7 BND OTU B3:4/8 EOR
%   I:1.0/7  LINE_4_START_BUTTON %
%   B3:4/7  LINE_4_FEED_START %
%   B3:4/8  LINE_4_FEED_STOPPED %

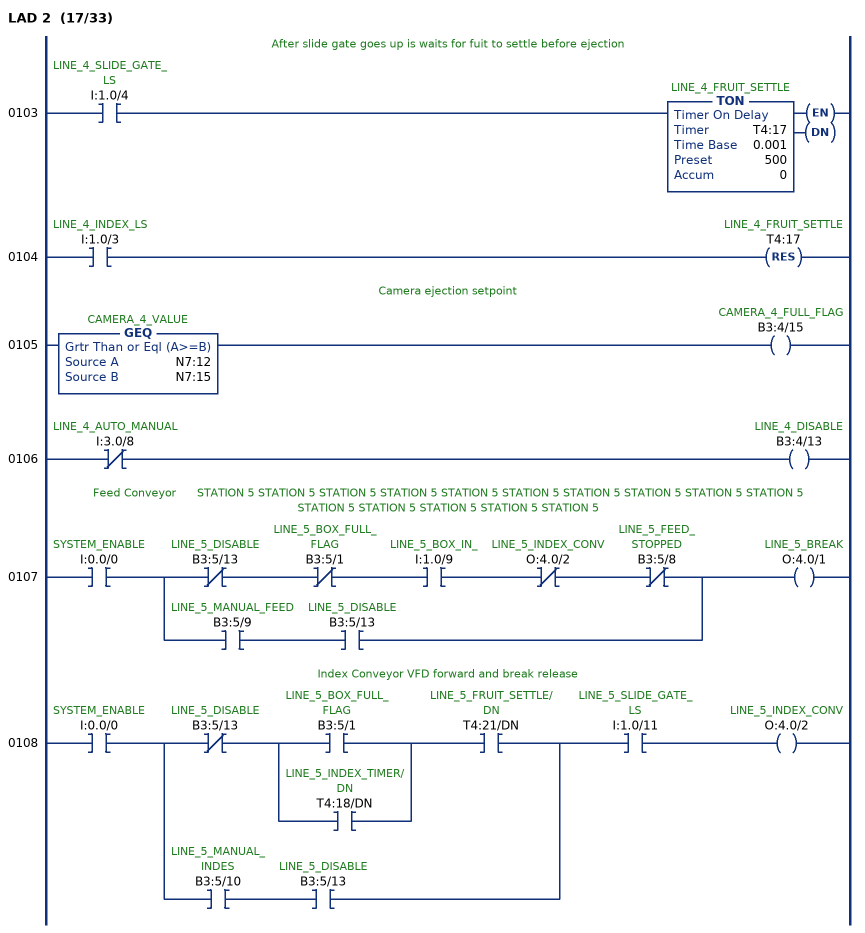
% Rung: 103 %
% After slide gate goes up is waits for fuit to settle before ejection %
SOR XIC I:1.0/4 TON T4:17 0.001 500 0 EOR
%   I:1.0/4  LINE_4_SLIDE_GATE_LS %
%   T4:17  LINE_4_FRUIT_SETTLE %
% Rung: 104 %
SOR XIC I:1.0/3 RES T4:17 EOR
%   I:1.0/3  LINE_4_INDEX_LS %
%   T4:17  LINE_4_FRUIT_SETTLE %
% Rung: 105 %
% Camera ejection setpoint %
SOR GEQ N7:12 N7:15 OTE B3:4/15 EOR
%   N7:12  CAMERA_4_VALUE %
%   N7:15  CAMERA_4_EJECT %
%   B3:4/15  CAMERA_4_FULL_FLAG %
% Rung: 106 %
SOR XIO I:3.0/8 OTE B3:4/13 EOR
%   I:3.0/8  LINE_4_AUTO_MANUAL %
%   B3:4/13  LINE_4_DISABLE %
% Rung: 107 %
% Feed Conveyor      STATION 5 STATION 5 STATION 5 STATION 5 STATION 5 STATION 5 STATION 5 STATION 5 STATION 5 STATION 5 STATION 5 STATION 5 STATION 5 STATION 5 STATION 5 %
SOR XIC I:0.0/0 BST XIO B3:5/13 XIO B3:5/1 XIC I:1.0/9 XIO O:4.0/2 XIO B3:5/8 NXB XIC B3:5/9 XIC B3:5/13 BND OTE O:4.0/1 EOR
%   I:0.0/0  SYSTEM_ENABLE %
%   B3:5/13  LINE_5_DISABLE %
%   B3:5/1  LINE_5_BOX_FULL_FLAG %
%   I:1.0/9  LINE_5_BOX_IN_ %
%   O:4.0/2  LINE_5_INDEX_CONV %
%   B3:5/8  LINE_5_FEED_STOPPED %
%   B3:5/9  LINE_5_MANUAL_FEED %
%   O:4.0/1  LINE_5_BREAK %
% Rung: 108 %
% Index Conveyor VFD forward and break release %
SOR XIC I:0.0/0 BST XIO B3:5/13 BST XIC B3:5/1 NXB XIC T4:18/DN BND XIC T4:21/DN NXB XIC B3:5/10 XIC B3:5/13 BND XIC I:1.0/11 OTE O:4.0/2 EOR
%   I:0.0/0  SYSTEM_ENABLE %
%   B3:5/13  LINE_5_DISABLE %
%   B3:5/1  LINE_5_BOX_FULL_FLAG %
%   T4:18  LINE_5_INDEX_TIMER %
%   T4:21  LINE_5_FRUIT_SETTLE %
%   B3:5/10  LINE_5_MANUAL_INDES %
%   I:1.0/11  LINE_5_SLIDE_GATE_LS %
%   O:4.0/2  LINE_5_INDEX_CONV %

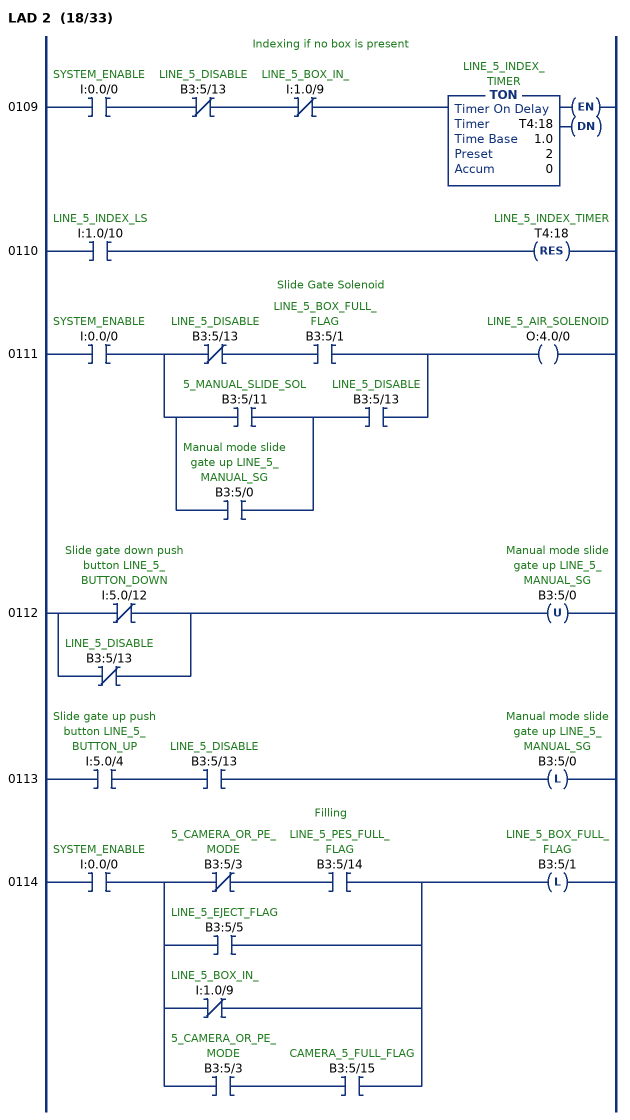
% Rung: 109 %
% Indexing if no box is present %
SOR XIC I:0.0/0 XIO B3:5/13 XIO I:1.0/9 TON T4:18 1.0 2 0 EOR
%   I:0.0/0  SYSTEM_ENABLE %
%   B3:5/13  LINE_5_DISABLE %
%   I:1.0/9  LINE_5_BOX_IN_ %
%   T4:18  LINE_5_INDEX_TIMER %
% Rung: 110 %
SOR XIC I:1.0/10 RES T4:18 EOR
%   I:1.0/10  LINE_5_INDEX_LS %
%   T4:18  LINE_5_INDEX_TIMER %
% Rung: 111 %
% Slide Gate Solenoid %
SOR XIC I:0.0/0 BST XIO B3:5/13 XIC B3:5/1 NXB BST XIC B3:5/11 NXB XIC B3:5/0 BND XIC B3:5/13 BND OTE O:4.0/0 EOR
%   I:0.0/0  SYSTEM_ENABLE %
%   B3:5/13  LINE_5_DISABLE %
%   B3:5/1  LINE_5_BOX_FULL_FLAG %
%   B3:5/11  5_MANUAL_SLIDE_SOL %
%   B3:5/0  LINE_5_MANUAL_SG  "Manual mode slide gate up" %
%   O:4.0/0  LINE_5_AIR_SOLENOID %
% Rung: 112 %
SOR BST XIO I:5.0/12 NXB XIO B3:5/13 BND OTU B3:5/0 EOR
%   I:5.0/12  LINE_5_BUTTON_DOWN  "Slide gate down push button" %
%   B3:5/13  LINE_5_DISABLE %
%   B3:5/0  LINE_5_MANUAL_SG  "Manual mode slide gate up" %
% Rung: 113 %
SOR XIC I:5.0/4 XIC B3:5/13 OTL B3:5/0 EOR
%   I:5.0/4  LINE_5_BUTTON_UP  "Slide gate up push button" %
%   B3:5/13  LINE_5_DISABLE %
%   B3:5/0  LINE_5_MANUAL_SG  "Manual mode slide gate up" %
% Rung: 114 %
% Filling %
SOR XIC I:0.0/0 BST XIO B3:5/3 XIC B3:5/14 NXB BST XIC B3:5/5 NXB BST XIO I:1.0/9 NXB XIC B3:5/3 XIC B3:5/15 BND BND BND OTL B3:5/1 EOR
%   I:0.0/0  SYSTEM_ENABLE %
%   B3:5/3  5_CAMERA_OR_PE_MODE %
%   B3:5/14  LINE_5_PES_FULL_FLAG %
%   B3:5/5  LINE_5_EJECT_FLAG %
%   I:1.0/9  LINE_5_BOX_IN_ %
%   B3:5/15  CAMERA_5_FULL_FLAG %
%   B3:5/1  LINE_5_BOX_FULL_FLAG %

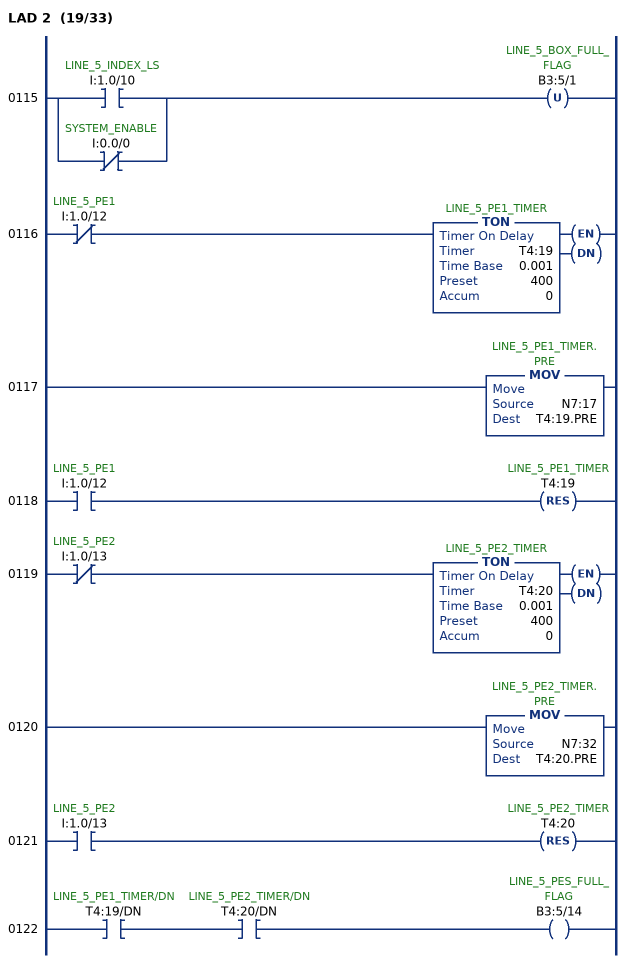
% Rung: 115 %
SOR BST XIC I:1.0/10 NXB XIO I:0.0/0 BND OTU B3:5/1 EOR
%   I:1.0/10  LINE_5_INDEX_LS %
%   I:0.0/0  SYSTEM_ENABLE %
%   B3:5/1  LINE_5_BOX_FULL_FLAG %
% Rung: 116 %
SOR XIO I:1.0/12 TON T4:19 0.001 400 0 EOR
%   I:1.0/12  LINE_5_PE1 %
%   T4:19  LINE_5_PE1_TIMER %
% Rung: 117 %
SOR MOV N7:17 T4:19.PRE EOR
%   N7:17  LINE_5_PE1_TIME_MOV %
%   T4:19  LINE_5_PE1_TIMER %
% Rung: 118 %
SOR XIC I:1.0/12 RES T4:19 EOR
%   I:1.0/12  LINE_5_PE1 %
%   T4:19  LINE_5_PE1_TIMER %
% Rung: 119 %
SOR XIO I:1.0/13 TON T4:20 0.001 400 0 EOR
%   I:1.0/13  LINE_5_PE2 %
%   T4:20  LINE_5_PE2_TIMER %
% Rung: 120 %
SOR MOV N7:32 T4:20.PRE EOR
%   N7:32  LINE_5_PE2_TIME_MOV %
%   T4:20  LINE_5_PE2_TIMER %
% Rung: 121 %
SOR XIC I:1.0/13 RES T4:20 EOR
%   I:1.0/13  LINE_5_PE2 %
%   T4:20  LINE_5_PE2_TIMER %
% Rung: 122 %
SOR XIC T4:19/DN XIC T4:20/DN OTE B3:5/14 EOR
%   T4:19  LINE_5_PE1_TIMER %
%   T4:20  LINE_5_PE2_TIMER %
%   B3:5/14  LINE_5_PES_FULL_FLAG %

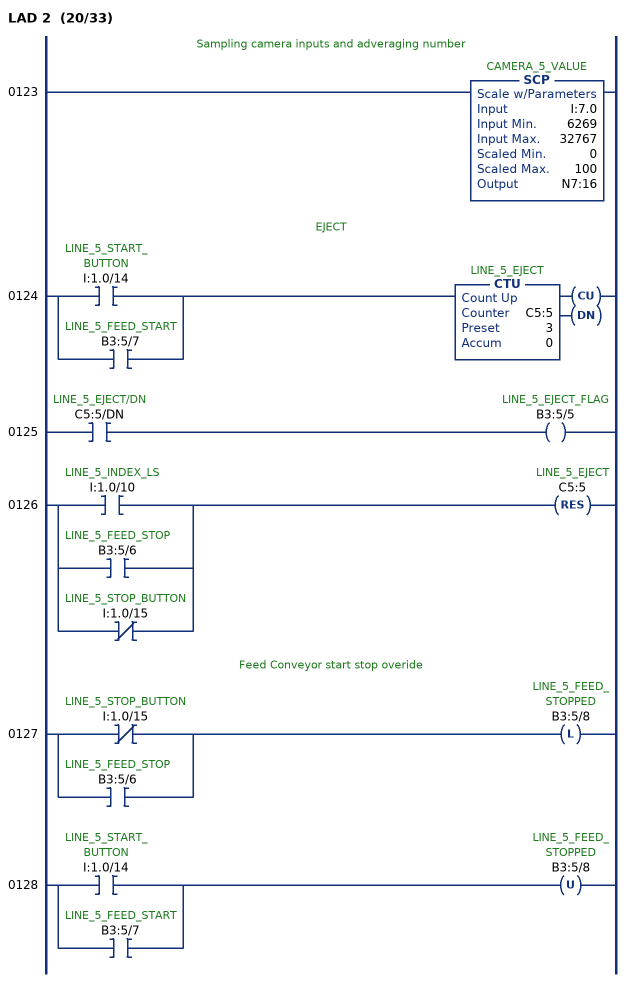
% Rung: 123 %
% Sampling camera inputs and adveraging number %
SOR SCP I:7.0 6269 32767 0 100 N7:16 EOR
%   N7:16  CAMERA_5_VALUE %
% Rung: 124 %
% EJECT %
SOR BST XIC I:1.0/14 NXB XIC B3:5/7 BND CTU C5:5 3 0 EOR
%   I:1.0/14  LINE_5_START_BUTTON %
%   B3:5/7  LINE_5_FEED_START %
%   C5:5  LINE_5_EJECT %
% Rung: 125 %
SOR XIC C5:5/DN OTE B3:5/5 EOR
%   C5:5  LINE_5_EJECT %
%   B3:5/5  LINE_5_EJECT_FLAG %
% Rung: 126 %
SOR BST XIC I:1.0/10 NXB BST XIC B3:5/6 NXB XIO I:1.0/15 BND BND RES C5:5 EOR
%   I:1.0/10  LINE_5_INDEX_LS %
%   B3:5/6  LINE_5_FEED_STOP %
%   I:1.0/15  LINE_5_STOP_BUTTON %
%   C5:5  LINE_5_EJECT %
% Rung: 127 %
% Feed Conveyor start stop overide %
SOR BST XIO I:1.0/15 NXB XIC B3:5/6 BND OTL B3:5/8 EOR
%   I:1.0/15  LINE_5_STOP_BUTTON %
%   B3:5/6  LINE_5_FEED_STOP %
%   B3:5/8  LINE_5_FEED_STOPPED %
% Rung: 128 %
SOR BST XIC I:1.0/14 NXB XIC B3:5/7 BND OTU B3:5/8 EOR
%   I:1.0/14  LINE_5_START_BUTTON %
%   B3:5/7  LINE_5_FEED_START %
%   B3:5/8  LINE_5_FEED_STOPPED %

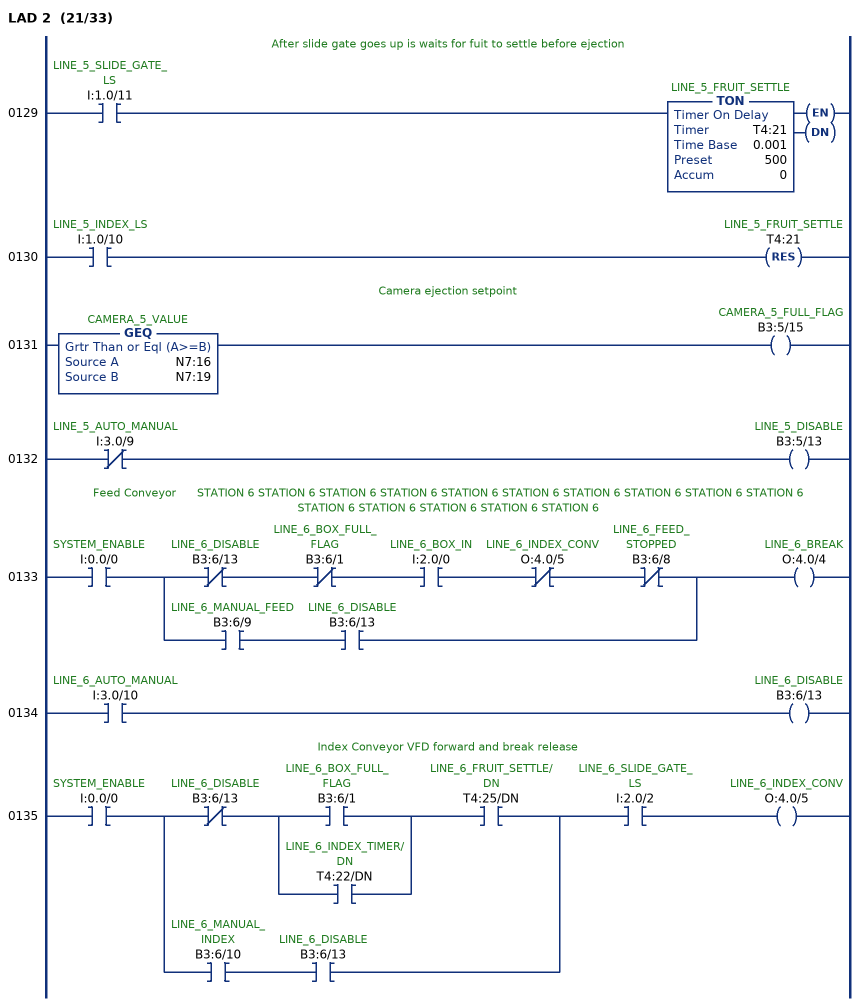
% Rung: 129 %
% After slide gate goes up is waits for fuit to settle before ejection %
SOR XIC I:1.0/11 TON T4:21 0.001 500 0 EOR
%   I:1.0/11  LINE_5_SLIDE_GATE_LS %
%   T4:21  LINE_5_FRUIT_SETTLE %
% Rung: 130 %
SOR XIC I:1.0/10 RES T4:21 EOR
%   I:1.0/10  LINE_5_INDEX_LS %
%   T4:21  LINE_5_FRUIT_SETTLE %
% Rung: 131 %
% Camera ejection setpoint %
SOR GEQ N7:16 N7:19 OTE B3:5/15 EOR
%   N7:16  CAMERA_5_VALUE %
%   N7:19  CAMERA_5_EJECT %
%   B3:5/15  CAMERA_5_FULL_FLAG %
% Rung: 132 %
SOR XIO I:3.0/9 OTE B3:5/13 EOR
%   I:3.0/9  LINE_5_AUTO_MANUAL %
%   B3:5/13  LINE_5_DISABLE %
% Rung: 133 %
% Feed Conveyor      STATION 6 STATION 6 STATION 6 STATION 6 STATION 6 STATION 6 STATION 6 STATION 6 STATION 6 STATION 6 STATION 6 STATION 6 STATION 6 STATION 6 STATION 6 %
SOR XIC I:0.0/0 BST XIO B3:6/13 XIO B3:6/1 XIC I:2.0/0 XIO O:4.0/5 XIO B3:6/8 NXB XIC B3:6/9 XIC B3:6/13 BND OTE O:4.0/4 EOR
%   I:0.0/0  SYSTEM_ENABLE %
%   B3:6/13  LINE_6_DISABLE %
%   B3:6/1  LINE_6_BOX_FULL_FLAG %
%   I:2.0/0  LINE_6_BOX_IN %
%   O:4.0/5  LINE_6_INDEX_CONV %
%   B3:6/8  LINE_6_FEED_STOPPED %
%   B3:6/9  LINE_6_MANUAL_FEED %
%   O:4.0/4  LINE_6_BREAK %
% Rung: 134 %
SOR XIC I:3.0/10 OTE B3:6/13 EOR
%   I:3.0/10  LINE_6_AUTO_MANUAL %
%   B3:6/13  LINE_6_DISABLE %
% Rung: 135 %
% Index Conveyor VFD forward and break release %
SOR XIC I:0.0/0 BST XIO B3:6/13 BST XIC B3:6/1 NXB XIC T4:22/DN BND XIC T4:25/DN NXB XIC B3:6/10 XIC B3:6/13 BND XIC I:2.0/2 OTE O:4.0/5 EOR
%   I:0.0/0  SYSTEM_ENABLE %
%   B3:6/13  LINE_6_DISABLE %
%   B3:6/1  LINE_6_BOX_FULL_FLAG %
%   T4:22  LINE_6_INDEX_TIMER %
%   T4:25  LINE_6_FRUIT_SETTLE %
%   B3:6/10  LINE_6_MANUAL_INDEX %
%   I:2.0/2  LINE_6_SLIDE_GATE_LS %
%   O:4.0/5  LINE_6_INDEX_CONV %

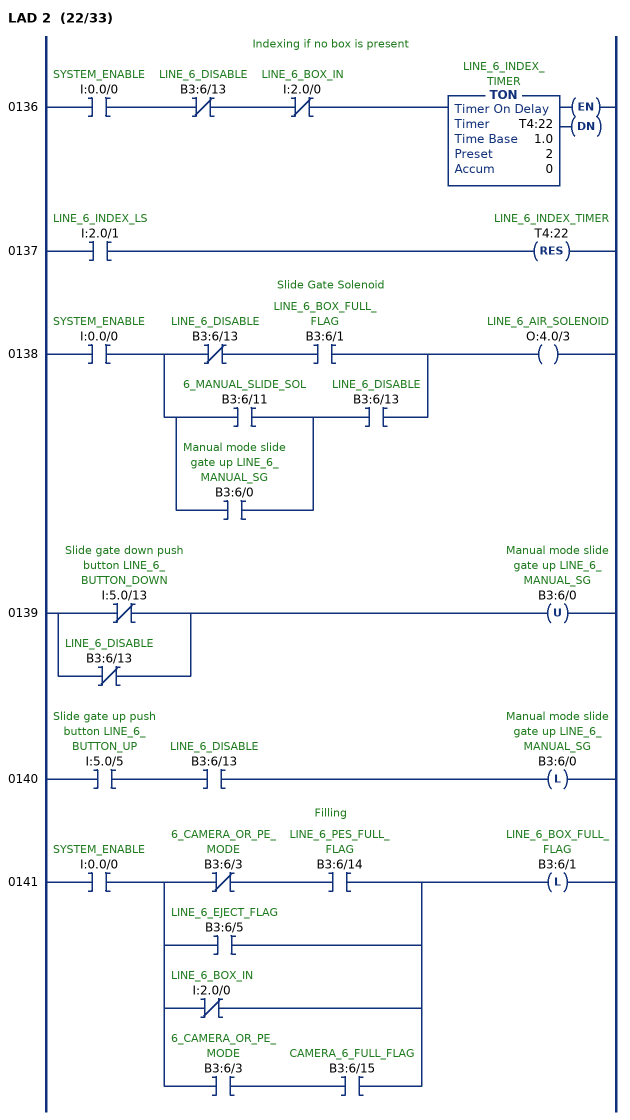
% Rung: 136 %
% Indexing if no box is present %
SOR XIC I:0.0/0 XIO B3:6/13 XIO I:2.0/0 TON T4:22 1.0 2 0 EOR
%   I:0.0/0  SYSTEM_ENABLE %
%   B3:6/13  LINE_6_DISABLE %
%   I:2.0/0  LINE_6_BOX_IN %
%   T4:22  LINE_6_INDEX_TIMER %
% Rung: 137 %
SOR XIC I:2.0/1 RES T4:22 EOR
%   I:2.0/1  LINE_6_INDEX_LS %
%   T4:22  LINE_6_INDEX_TIMER %
% Rung: 138 %
% Slide Gate Solenoid %
SOR XIC I:0.0/0 BST XIO B3:6/13 XIC B3:6/1 NXB BST XIC B3:6/11 NXB XIC B3:6/0 BND XIC B3:6/13 BND OTE O:4.0/3 EOR
%   I:0.0/0  SYSTEM_ENABLE %
%   B3:6/13  LINE_6_DISABLE %
%   B3:6/1  LINE_6_BOX_FULL_FLAG %
%   B3:6/11  6_MANUAL_SLIDE_SOL %
%   B3:6/0  LINE_6_MANUAL_SG  "Manual mode slide gate up" %
%   O:4.0/3  LINE_6_AIR_SOLENOID %
% Rung: 139 %
SOR BST XIO I:5.0/13 NXB XIO B3:6/13 BND OTU B3:6/0 EOR
%   I:5.0/13  LINE_6_BUTTON_DOWN  "Slide gate down push button" %
%   B3:6/13  LINE_6_DISABLE %
%   B3:6/0  LINE_6_MANUAL_SG  "Manual mode slide gate up" %
% Rung: 140 %
SOR XIC I:5.0/5 XIC B3:6/13 OTL B3:6/0 EOR
%   I:5.0/5  LINE_6_BUTTON_UP  "Slide gate up push button" %
%   B3:6/13  LINE_6_DISABLE %
%   B3:6/0  LINE_6_MANUAL_SG  "Manual mode slide gate up" %
% Rung: 141 %
% Filling %
SOR XIC I:0.0/0 BST XIO B3:6/3 XIC B3:6/14 NXB BST XIC B3:6/5 NXB BST XIO I:2.0/0 NXB XIC B3:6/3 XIC B3:6/15 BND BND BND OTL B3:6/1 EOR
%   I:0.0/0  SYSTEM_ENABLE %
%   B3:6/3  6_CAMERA_OR_PE_MODE %
%   B3:6/14  LINE_6_PES_FULL_FLAG %
%   B3:6/5  LINE_6_EJECT_FLAG %
%   I:2.0/0  LINE_6_BOX_IN %
%   B3:6/15  CAMERA_6_FULL_FLAG %
%   B3:6/1  LINE_6_BOX_FULL_FLAG %

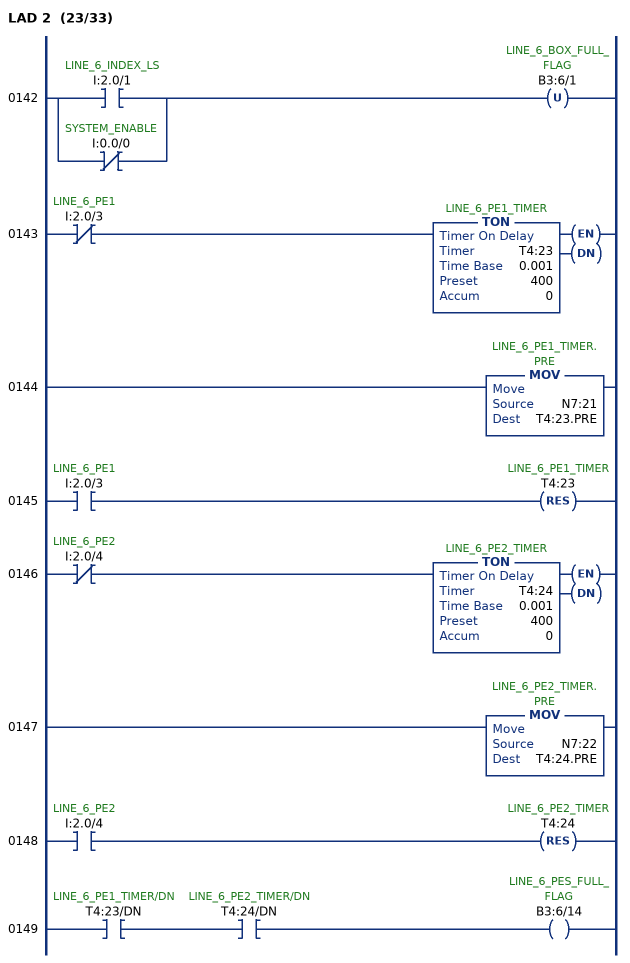
% Rung: 142 %
SOR BST XIC I:2.0/1 NXB XIO I:0.0/0 BND OTU B3:6/1 EOR
%   I:2.0/1  LINE_6_INDEX_LS %
%   I:0.0/0  SYSTEM_ENABLE %
%   B3:6/1  LINE_6_BOX_FULL_FLAG %
% Rung: 143 %
SOR XIO I:2.0/3 TON T4:23 0.001 400 0 EOR
%   I:2.0/3  LINE_6_PE1 %
%   T4:23  LINE_6_PE1_TIMER %
% Rung: 144 %
SOR MOV N7:21 T4:23.PRE EOR
%   N7:21  LINE_6_PE1_TIME_MOV %
%   T4:23  LINE_6_PE1_TIMER %
% Rung: 145 %
SOR XIC I:2.0/3 RES T4:23 EOR
%   I:2.0/3  LINE_6_PE1 %
%   T4:23  LINE_6_PE1_TIMER %
% Rung: 146 %
SOR XIO I:2.0/4 TON T4:24 0.001 400 0 EOR
%   I:2.0/4  LINE_6_PE2 %
%   T4:24  LINE_6_PE2_TIMER %
% Rung: 147 %
SOR MOV N7:22 T4:24.PRE EOR
%   N7:22  LINE_6_PE2_TIME_MOV %
%   T4:24  LINE_6_PE2_TIMER %
% Rung: 148 %
SOR XIC I:2.0/4 RES T4:24 EOR
%   I:2.0/4  LINE_6_PE2 %
%   T4:24  LINE_6_PE2_TIMER %
% Rung: 149 %
SOR XIC T4:23/DN XIC T4:24/DN OTE B3:6/14 EOR
%   T4:23  LINE_6_PE1_TIMER %
%   T4:24  LINE_6_PE2_TIMER %
%   B3:6/14  LINE_6_PES_FULL_FLAG %

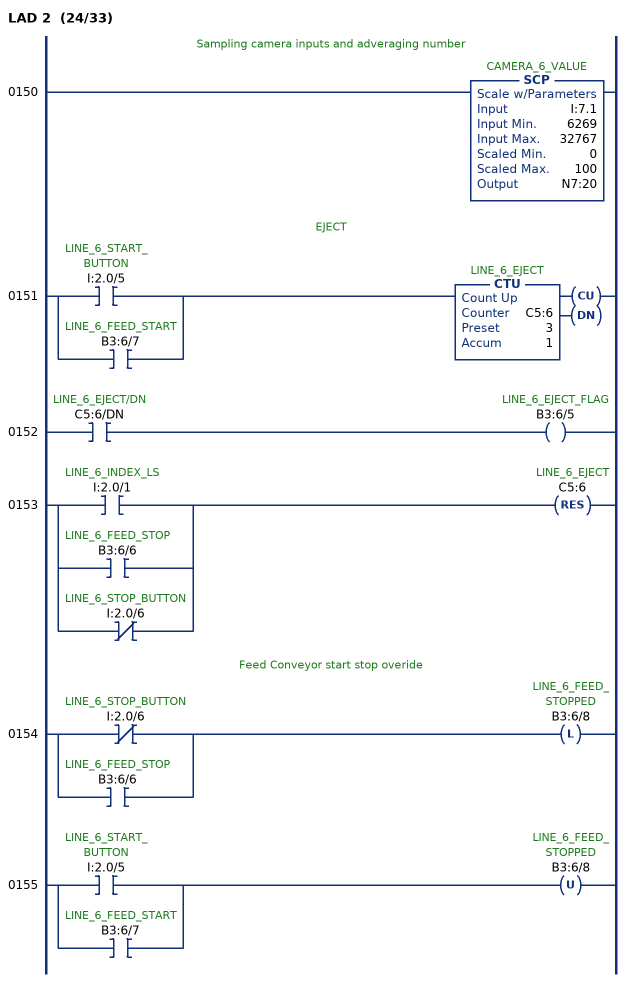
% Rung: 150 %
% Sampling camera inputs and adveraging number %
SOR SCP I:7.1 6269 32767 0 100 N7:20 EOR
%   N7:20  CAMERA_6_VALUE %
% Rung: 151 %
% EJECT %
SOR BST XIC I:2.0/5 NXB XIC B3:6/7 BND CTU C5:6 3 1 EOR
%   I:2.0/5  LINE_6_START_BUTTON %
%   B3:6/7  LINE_6_FEED_START %
%   C5:6  LINE_6_EJECT %
% Rung: 152 %
SOR XIC C5:6/DN OTE B3:6/5 EOR
%   C5:6  LINE_6_EJECT %
%   B3:6/5  LINE_6_EJECT_FLAG %
% Rung: 153 %
SOR BST XIC I:2.0/1 NXB BST XIC B3:6/6 NXB XIO I:2.0/6 BND BND RES C5:6 EOR
%   I:2.0/1  LINE_6_INDEX_LS %
%   B3:6/6  LINE_6_FEED_STOP %
%   I:2.0/6  LINE_6_STOP_BUTTON %
%   C5:6  LINE_6_EJECT %
% Rung: 154 %
% Feed Conveyor start stop overide %
SOR BST XIO I:2.0/6 NXB XIC B3:6/6 BND OTL B3:6/8 EOR
%   I:2.0/6  LINE_6_STOP_BUTTON %
%   B3:6/6  LINE_6_FEED_STOP %
%   B3:6/8  LINE_6_FEED_STOPPED %
% Rung: 155 %
SOR BST XIC I:2.0/5 NXB XIC B3:6/7 BND OTU B3:6/8 EOR
%   I:2.0/5  LINE_6_START_BUTTON %
%   B3:6/7  LINE_6_FEED_START %
%   B3:6/8  LINE_6_FEED_STOPPED %

